C09150=1146.700,365.761,-82.220,-176.299,9.450,148.853
C09151=1146.704,365.478,-82.179,-176.301,9.445,148.852
C09152=1146.709,365.195,-82.139,-176.305,9.440,148.852
C09153=1146.713,364.911,-82.098,-176.307,9.436,148.851
C09154=1146.718,364.628,-82.057,-176.311,9.431,148.851
C09155=1146.722,364.381,-82.022,-176.313,9.427,148.851
C09156=1146.726,364.133,-81.986,-176.316,9.423,148.850
C09157=1146.730,363.886,-81.950,-176.318,9.419,148.850
C09158=1146.734,363.638,-81.915,-176.321,9.415,148.850
C09159=1146.737,363.391,-81.879,-176.323,9.411,148.849
C09160=1146.741,363.144,-81.844,-176.326,9.406,148.849
C09161=1146.745,362.896,-81.808,-176.329,9.402,148.849
C09162=1146.749,362.648,-81.773,-176.331,9.399,148.848
C09163=1146.753,362.401,-81.738,-176.334,9.394,148.848
C09164=1146.757,362.154,-81.703,-176.336,9.390,148.848
C09165=1146.761,361.906,-81.667,-176.339,9.386,148.847
C09166=1146.764,361.659,-81.632,-176.341,9.383,148.847
C09167=1146.768,361.411,-81.597,-176.344,9.379,148.847
C09168=1146.773,361.164,-81.562,-176.347,9.374,148.846
C09169=1146.776,360.917,-81.526,-176.350,9.370,148.846
C09170=1146.780,360.669,-81.490,-176.352,9.367,148.846
C09171=1146.784,360.421,-81.456,-176.354,9.362,148.845
C09172=1146.788,360.174,-81.420,-176.357,9.358,148.845
C09173=1146.792,359.927,-81.385,-176.359,9.355,148.845
C09174=1146.796,359.678,-81.350,-176.362,9.350,148.844
C09175=1146.800,359.432,-81.315,-176.365,9.346,148.844
C09176=1146.804,359.184,-81.280,-176.368,9.342,148.844
C09177=1146.808,358.936,-81.245,-176.369,9.339,148.843
C09178=1146.812,358.689,-81.209,-176.372,9.335,148.843
C09179=1146.816,358.441,-81.175,-176.375,9.330,148.842
C09180=1146.820,358.194,-81.139,-176.377,9.327,148.842
C09181=1146.823,357.947,-81.105,-176.380,9.323,148.842
C09182=1146.827,357.699,-81.070,-176.383,9.318,148.842
C09183=1146.831,357.451,-81.035,-176.385,9.315,148.841
C09184=1146.835,357.204,-81.000,-176.387,9.311,148.841
C09185=1146.839,356.956,-80.965,-176.390,9.306,148.840
C09186=1146.843,356.708,-80.929,-176.392,9.303,148.840
C09187=1146.847,356.461,-80.895,-176.395,9.299,148.840
C09188=1146.850,356.214,-80.860,-176.397,9.295,148.840
C09189=1146.855,355.966,-80.825,-176.400,9.291,148.839
C09190=1146.859,355.719,-80.790,-176.402,9.287,148.839
C09191=1146.863,355.471,-80.755,-176.405,9.284,148.839
C09192=1146.867,355.223,-80.720,-176.407,9.279,148.838
C09193=1146.870,354.976,-80.685,-176.410,9.275,148.838
C09194=1146.875,354.729,-80.651,-176.413,9.272,148.838
C09195=1146.879,354.481,-80.616,-176.415,9.268,148.837
C09196=1146.882,354.233,-80.581,-176.417,9.264,148.837
C09197=1146.886,353.986,-80.547,-176.420,9.260,148.837
C09198=1146.890,353.738,-80.512,-176.423,9.256,148.836
C09199=1146.894,353.491,-80.477,-176.425,9.252,148.836
C09200=1146.898,353.243,-80.442,-176.428,9.248,148.836
C09201=1146.902,352.996,-80.408,-176.431,9.244,148.835
C09202=1146.906,352.748,-80.373,-176.432,9.240,148.835
C09203=1146.910,352.501,-80.338,-176.435,9.236,148.835
C09204=1146.914,352.253,-80.304,-176.437,9.233,148.834
C09205=1146.918,352.006,-80.269,-176.440,9.229,148.834
C09206=1146.922,351.758,-80.234,-176.443,9.225,148.834
C09207=1146.926,351.511,-80.201,-176.445,9.221,148.833
C09208=1146.930,351.263,-80.165,-176.448,9.217,148.833
C09209=1146.934,351.016,-80.131,-176.450,9.213,148.833
C09210=1146.937,350.768,-80.096,-176.453,9.209,148.832
C09211=1146.942,350.520,-80.062,-176.456,9.205,148.832
C09212=1146.946,350.272,-80.027,-176.458,9.202,148.832
C09213=1146.950,350.025,-79.993,-176.460,9.198,148.832
C09214=1146.954,349.777,-79.958,-176.463,9.194,148.831
C09215=1146.958,349.530,-79.924,-176.465,9.190,148.831
C09216=1146.962,349.282,-79.890,-176.468,9.186,148.831
C09217=1146.966,349.034,-79.855,-176.470,9.183,148.830
C09218=1146.969,348.787,-79.821,-176.473,9.178,148.830
C09219=1146.974,348.539,-79.786,-176.475,9.175,148.830
C09220=1146.978,348.292,-79.753,-176.478,9.171,148.830
C09221=1146.982,348.044,-79.718,-176.480,9.167,148.829
C09222=1146.986,347.797,-79.684,-176.483,9.163,148.829
C09223=1146.990,347.549,-79.649,-176.486,9.159,148.829
C09224=1146.993,347.302,-79.615,-176.488,9.155,148.828
C09225=1146.997,347.053,-79.580,-176.491,9.151,148.828
C09226=1147.001,346.806,-79.546,-176.493,9.148,148.828
C09227=1147.006,346.558,-79.513,-176.496,9.144,148.827
C09228=1147.009,346.311,-79.479,-176.498,9.140,148.827
C09229=1147.014,346.063,-79.444,-176.501,9.136,148.827
C09230=1147.018,345.816,-79.410,-176.503,9.132,148.826
C09231=1147.022,345.568,-79.375,-176.506,9.129,148.826
C09232=1147.026,345.321,-79.341,-176.509,9.125,148.826
C09233=1147.030,345.072,-79.307,-176.510,9.121,148.826
C09234=1147.034,344.825,-79.273,-176.513,9.117,148.825
C09235=1147.037,344.578,-79.240,-176.516,9.114,148.825
C09236=1147.042,344.329,-79.205,-176.519,9.110,148.825
C09237=1147.046,344.082,-79.172,-176.520,9.106,148.824
C09238=1147.050,343.835,-79.137,-176.523,9.102,148.824
C09239=1147.053,343.587,-79.103,-176.526,9.098,148.824
C09240=1147.058,343.339,-79.070,-176.528,9.094,148.824
C09241=1147.062,343.092,-79.035,-176.531,9.090,148.823
C09242=1147.066,342.844,-79.001,-176.533,9.087,148.823
C09243=1147.069,342.596,-78.968,-176.536,9.083,148.823
C09244=1147.074,342.349,-78.933,-176.538,9.079,148.822
C09245=1147.078,342.101,-78.900,-176.541,9.075,148.822
C09246=1147.081,341.853,-78.866,-176.544,9.072,148.822
C09247=1147.086,341.606,-78.832,-176.546,9.068,148.822
C09248=1147.090,341.358,-78.798,-176.548,9.064,148.821
C09249=1147.094,341.111,-78.765,-176.551,9.060,148.821
C09250=1147.098,340.862,-78.730,-176.554,9.057,148.821
C09251=1147.102,340.615,-78.697,-176.556,9.053,148.821
C09252=1147.106,340.367,-78.663,-176.558,9.049,148.820
C09253=1147.110,340.120,-78.630,-176.561,9.045,148.820
C09254=1147.114,339.871,-78.595,-176.564,9.041,148.820
C09255=1147.119,339.592,-78.558,-176.567,9.037,148.819
C09256=1147.124,339.311,-78.519,-176.570,9.033,148.819
C09257=1147.128,339.031,-78.481,-176.573,9.028,148.819
C09258=1147.132,338.750,-78.443,-176.575,9.024,148.819
C09259=1147.136,338.503,-78.410,-176.578,9.021,148.818
C09260=1147.140,338.255,-78.376,-176.581,9.017,148.818
C09261=1147.144,338.008,-78.343,-176.583,9.013,148.818
C09262=1147.149,337.760,-78.309,-176.585,9.009,148.817
C09263=1147.153,337.512,-78.275,-176.588,9.005,148.817
C09264=1147.157,337.264,-78.242,-176.591,9.002,148.817
C09265=1147.161,337.016,-78.209,-176.594,8.998,148.817
C09266=1147.165,336.769,-78.175,-176.596,8.995,148.817
C09267=1147.169,336.522,-78.141,-176.598,8.990,148.816
C09268=1147.172,336.273,-78.108,-176.601,8.987,148.816
C09269=1147.176,336.025,-78.075,-176.604,8.983,148.816
C09270=1147.181,335.778,-78.040,-176.606,8.980,148.815
C09271=1147.185,335.530,-78.007,-176.608,8.976,148.815
C09272=1147.189,335.283,-77.974,-176.611,8.972,148.815
C09273=1147.193,335.035,-77.941,-176.613,8.969,148.815
C09274=1147.198,334.787,-77.908,-176.616,8.965,148.814
C09275=1147.201,334.539,-77.874,-176.618,8.961,148.814
C09276=1147.205,334.292,-77.840,-176.621,8.957,148.814
C09277=1147.209,334.044,-77.807,-176.624,8.954,148.814
C09278=1147.213,333.796,-77.774,-176.627,8.950,148.813
C09279=1147.217,333.548,-77.741,-176.629,8.947,148.813
C09280=1147.222,333.301,-77.708,-176.631,8.942,148.813
C09281=1147.226,333.053,-77.675,-176.634,8.939,148.813
C09282=1147.230,332.805,-77.641,-176.637,8.935,148.812
C09283=1147.234,332.557,-77.608,-176.639,8.932,148.812
C09284=1147.237,332.309,-77.575,-176.642,8.928,148.812
C09285=1147.242,332.061,-77.542,-176.644,8.924,148.812
C09286=1147.246,331.814,-77.508,-176.647,8.920,148.812
C09287=1147.250,331.566,-77.475,-176.649,8.917,148.811
C09288=1147.253,331.318,-77.443,-176.652,8.913,148.811
C09289=1147.257,331.071,-77.410,-176.655,8.910,148.811
C09290=1147.262,330.823,-77.376,-176.657,8.906,148.811
C09291=1147.266,330.575,-77.343,-176.659,8.902,148.810
C09292=1147.270,330.327,-77.310,-176.662,8.899,148.810
C09293=1147.274,330.080,-77.277,-176.665,8.895,148.810
C09294=1147.278,329.832,-77.244,-176.667,8.891,148.810
C09295=1147.283,329.584,-77.211,-176.670,8.887,148.809
C09296=1147.287,329.336,-77.178,-176.672,8.884,148.809
C09297=1147.290,329.089,-77.146,-176.675,8.880,148.809
C09298=1147.294,328.841,-77.112,-176.677,8.877,148.809
C09299=1147.298,328.593,-77.079,-176.680,8.872,148.809
C09300=1147.303,328.345,-77.046,-176.683,8.869,148.808
C09301=1147.307,328.097,-77.014,-176.685,8.866,148.808
C09302=1147.310,327.850,-76.981,-176.688,8.862,148.808
C09303=1147.315,327.602,-76.948,-176.690,8.859,148.808
C09304=1147.319,327.354,-76.915,-176.693,8.855,148.807
C09305=1147.323,327.106,-76.882,-176.696,8.851,148.807
C09306=1147.327,326.858,-76.849,-176.698,8.847,148.807
C09307=1147.331,326.611,-76.817,-176.701,8.844,148.807
C09308=1147.335,326.362,-76.784,-176.703,8.841,148.807
C09309=1147.339,326.115,-76.751,-176.706,8.837,148.806
C09310=1147.343,325.867,-76.719,-176.708,8.833,148.806
C09311=1147.347,325.619,-76.686,-176.711,8.829,148.806
C09312=1147.352,325.372,-76.653,-176.714,8.826,148.806
C09313=1147.356,325.123,-76.621,-176.716,8.822,148.806
C09314=1147.360,324.876,-76.588,-176.719,8.819,148.805
C09315=1147.364,324.628,-76.555,-176.721,8.815,148.805
C09316=1147.368,324.380,-76.523,-176.724,8.811,148.805
C09317=1147.372,324.132,-76.490,-176.726,8.808,148.805
C09318=1147.376,323.884,-76.458,-176.729,8.804,148.805
C09319=1147.380,323.636,-76.425,-176.732,8.801,148.804
C09320=1147.384,323.388,-76.393,-176.734,8.797,148.804
C09321=1147.388,323.141,-76.360,-176.737,8.793,148.804
C09322=1147.392,322.893,-76.328,-176.739,8.790,148.804
C09323=1147.396,322.646,-76.295,-176.742,8.786,148.803
C09324=1147.401,322.397,-76.262,-176.744,8.783,148.803
C09325=1147.404,322.150,-76.230,-176.747,8.779,148.803
C09326=1147.409,321.901,-76.197,-176.750,8.775,148.803
C09327=1147.412,321.653,-76.166,-176.752,8.772,148.803
C09328=1147.417,321.406,-76.132,-176.755,8.768,148.802
C09329=1147.421,321.158,-76.101,-176.757,8.765,148.802
C09330=1147.425,320.911,-76.068,-176.760,8.761,148.802
C09331=1147.429,320.663,-76.036,-176.762,8.757,148.802
C09332=1147.433,320.414,-76.004,-176.765,8.754,148.802
C09333=1147.437,320.167,-75.971,-176.768,8.750,148.801
C09334=1147.441,319.918,-75.939,-176.770,8.747,148.801
C09335=1147.445,319.671,-75.907,-176.773,8.744,148.801
C09336=1147.450,319.423,-75.875,-176.776,8.740,148.801
C09337=1147.453,319.175,-75.842,-176.778,8.736,148.801
C09338=1147.458,318.927,-75.810,-176.781,8.732,148.801
C09339=1147.461,318.679,-75.778,-176.783,8.729,148.800
C09340=1147.466,318.431,-75.746,-176.786,8.726,148.800
C09341=1147.470,318.184,-75.713,-176.788,8.722,148.800
C09342=1147.474,317.936,-75.681,-176.791,8.718,148.800
C09343=1147.478,317.687,-75.649,-176.793,8.715,148.800
C09344=1147.482,317.440,-75.617,-176.796,8.711,148.799
C09345=1147.487,317.192,-75.585,-176.799,8.708,148.799
C09346=1147.490,316.944,-75.553,-176.802,8.704,148.799
C09347=1147.495,316.695,-75.521,-176.804,8.701,148.799
C09348=1147.499,316.449,-75.488,-176.806,8.697,148.799
C09349=1147.503,316.201,-75.457,-176.809,8.693,148.799
C09350=1147.507,315.952,-75.424,-176.812,8.690,148.798
C09351=1147.511,315.704,-75.392,-176.814,8.687,148.798
C09352=1147.515,315.457,-75.361,-176.817,8.683,148.798
C09353=1147.519,315.209,-75.328,-176.820,8.680,148.798
C09354=1147.523,314.961,-75.297,-176.822,8.677,148.798
C09355=1147.527,314.713,-75.265,-176.825,8.672,148.798
C09356=1147.532,314.465,-75.233,-176.827,8.669,148.797
C09357=1147.536,314.217,-75.201,-176.830,8.666,148.797
C09358=1147.540,313.969,-75.169,-176.833,8.662,148.797
C09359=1147.545,313.692,-75.133,-176.836,8.658,148.797
C09360=1147.550,313.413,-75.098,-176.838,8.655,148.797
C09361=1147.554,313.136,-75.063,-176.841,8.651,148.797
C09362=1147.558,312.858,-75.027,-176.844,8.647,148.796
C09363=1147.563,312.610,-74.995,-176.847,8.643,148.796
C09364=1147.567,312.363,-74.963,-176.850,8.640,148.796
C09365=1147.571,312.115,-74.931,-176.852,8.636,148.796
C09366=1147.574,311.867,-74.899,-176.855,8.632,148.796
C09367=1147.579,311.619,-74.869,-176.857,8.629,148.796
C09368=1147.583,311.370,-74.836,-176.860,8.626,148.796
C09369=1147.588,311.123,-74.805,-176.863,8.622,148.795
C09370=1147.591,310.875,-74.773,-176.865,8.619,148.795
C09371=1147.596,310.626,-74.742,-176.867,8.615,148.795
C09372=1147.600,310.379,-74.710,-176.870,8.611,148.795
C09373=1147.604,310.131,-74.678,-176.873,8.608,148.795
C09374=1147.609,309.883,-74.646,-176.875,8.605,148.795
C09375=1147.613,309.635,-74.615,-176.878,8.602,148.794
C09376=1147.617,309.387,-74.584,-176.881,8.598,148.794
C09377=1147.621,309.139,-74.552,-176.883,8.595,148.794
C09378=1147.625,308.891,-74.521,-176.886,8.592,148.794
C09379=1147.629,308.643,-74.489,-176.889,8.587,148.794
C09380=1147.633,308.395,-74.457,-176.891,8.584,148.794
C09381=1147.637,308.147,-74.427,-176.894,8.581,148.794
C09382=1147.642,307.899,-74.394,-176.897,8.577,148.793
C09383=1147.646,307.651,-74.363,-176.899,8.574,148.793
C09384=1147.650,307.403,-74.332,-176.901,8.571,148.793
C09385=1147.654,307.156,-74.300,-176.905,8.567,148.793
C09386=1147.658,306.907,-74.269,-176.907,8.564,148.793
C09387=1147.663,306.660,-74.238,-176.909,8.560,148.793
C09388=1147.667,306.411,-74.206,-176.912,8.557,148.793
C09389=1147.671,306.164,-74.175,-176.915,8.553,148.793
C09390=1147.675,305.915,-74.144,-176.917,8.550,148.792
C09391=1147.679,305.668,-74.112,-176.920,8.547,148.792
C09392=1147.683,305.419,-74.081,-176.923,8.543,148.792
C09393=1147.688,305.172,-74.050,-176.925,8.540,148.792
C09394=1147.692,304.923,-74.019,-176.928,8.536,148.792
C09395=1147.696,304.675,-73.988,-176.930,8.534,148.792
C09396=1147.700,304.427,-73.956,-176.933,8.529,148.792
C09397=1147.705,304.179,-73.925,-176.936,8.526,148.791
C09398=1147.708,303.931,-73.893,-176.938,8.523,148.791
C09399=1147.713,303.683,-73.863,-176.941,8.519,148.791
C09400=1147.717,303.435,-73.832,-176.944,8.516,148.791
C09401=1147.720,303.187,-73.801,-176.946,8.513,148.791
C09402=1147.725,302.939,-73.770,-176.949,8.510,148.791
C09403=1147.729,302.691,-73.739,-176.952,8.506,148.791
C09404=1147.733,302.443,-73.707,-176.954,8.503,148.791
C09405=1147.738,302.195,-73.676,-176.957,8.499,148.791
C09406=1147.742,301.947,-73.645,-176.960,8.495,148.790
C09407=1147.747,301.699,-73.615,-176.963,8.492,148.790
C09408=1147.750,301.451,-73.583,-176.965,8.489,148.790
C09409=1147.754,301.203,-73.553,-176.967,8.486,148.790
C09410=1147.759,300.955,-73.522,-176.971,8.482,148.790
C09411=1147.763,300.706,-73.491,-176.973,8.479,148.790
C09412=1147.767,300.459,-73.460,-176.976,8.476,148.790
C09413=1147.771,300.210,-73.428,-176.978,8.473,148.790
C09414=1147.775,299.963,-73.398,-176.981,8.468,148.789
C09415=1147.780,299.715,-73.367,-176.984,8.466,148.789
C09416=1147.784,299.466,-73.336,-176.986,8.462,148.789
C09417=1147.788,299.218,-73.305,-176.988,8.459,148.789
C09418=1147.792,298.971,-73.275,-176.992,8.455,148.789
C09419=1147.796,298.722,-73.244,-176.994,8.452,148.789
C09420=1147.801,298.474,-73.213,-176.997,8.449,148.789
C09421=1147.805,298.226,-73.182,-176.999,8.446,148.789
C09422=1147.809,297.978,-73.152,-177.002,8.442,148.789
C09423=1147.813,297.730,-73.121,-177.005,8.439,148.789
C09424=1147.818,297.482,-73.090,-177.007,8.435,148.788
C09425=1147.822,297.233,-73.059,-177.010,8.433,148.788
C09426=1147.826,296.985,-73.029,-177.013,8.428,148.788
C09427=1147.830,296.737,-72.998,-177.015,8.425,148.788
C09428=1147.835,296.490,-72.967,-177.018,8.422,148.788
C09429=1147.838,296.241,-72.937,-177.020,8.419,148.788
C09430=1147.843,295.993,-72.906,-177.023,8.416,148.788
C09431=1147.847,295.746,-72.876,-177.026,8.412,148.788
C09432=1147.851,295.497,-72.845,-177.029,8.409,148.788
C09433=1147.855,295.249,-72.814,-177.031,8.406,148.788
C09434=1147.859,295.001,-72.784,-177.034,8.403,148.788
C09435=1147.864,294.753,-72.753,-177.037,8.399,148.787
C09436=1147.867,294.505,-72.723,-177.039,8.396,148.788
C09437=1147.872,294.256,-72.693,-177.042,8.392,148.787
C09438=1147.877,294.008,-72.662,-177.044,8.390,148.787
C09439=1147.881,293.761,-72.632,-177.047,8.386,148.787
C09440=1147.885,293.512,-72.601,-177.050,8.382,148.787
C09441=1147.888,293.265,-72.570,-177.052,8.379,148.787
C09442=1147.893,293.016,-72.540,-177.055,8.376,148.787
C09443=1147.897,292.768,-72.510,-177.058,8.373,148.787
C09444=1147.902,292.520,-72.479,-177.060,8.369,148.787
C09445=1147.905,292.271,-72.450,-177.063,8.366,148.787
C09446=1147.910,292.023,-72.419,-177.066,8.363,148.787
C09447=1147.914,291.776,-72.389,-177.068,8.360,148.787
C09448=1147.919,291.528,-72.358,-177.071,8.357,148.786
C09449=1147.923,291.280,-72.328,-177.074,8.353,148.786
C09450=1147.927,291.031,-72.297,-177.076,8.350,148.786
C09451=1147.931,290.783,-72.268,-177.079,8.347,148.786
C09452=1147.935,290.535,-72.238,-177.081,8.343,148.786
C09453=1147.939,290.287,-72.207,-177.084,8.340,148.786
C09454=1147.944,290.039,-72.177,-177.087,8.336,148.786
C09455=1147.948,289.791,-72.147,-177.090,8.333,148.786
C09456=1147.952,289.543,-72.117,-177.093,8.330,148.786
C09457=1147.956,289.294,-72.086,-177.095,8.327,148.786
C09458=1147.960,289.046,-72.056,-177.098,8.324,148.786
C09459=1147.964,288.798,-72.026,-177.100,8.321,148.786
C09460=1147.969,288.550,-71.996,-177.103,8.317,148.786
C09461=1147.973,288.302,-71.966,-177.106,8.314,148.786
C09462=1147.977,288.054,-71.936,-177.109,8.311,148.786
C09463=1147.982,287.778,-71.903,-177.111,8.307,148.785
C09464=1147.987,287.503,-71.869,-177.114,8.304,148.785
C09465=1147.992,287.228,-71.837,-177.118,8.300,148.785
C09466=1147.996,286.952,-71.803,-177.121,8.296,148.785
C09467=1148.001,286.703,-71.773,-177.123,8.293,148.785
C09468=1148.005,286.456,-71.743,-177.126,8.290,148.785
C09469=1148.009,286.208,-71.713,-177.128,8.287,148.785
C09470=1148.013,285.959,-71.684,-177.131,8.284,148.785
C09471=1148.018,285.711,-71.653,-177.133,8.281,148.785
C09472=1148.022,285.463,-71.624,-177.137,8.277,148.785
C09473=1148.026,285.215,-71.594,-177.139,8.274,148.785
C09474=1148.031,284.967,-71.563,-177.142,8.271,148.785
C09475=1148.035,284.719,-71.534,-177.144,8.267,148.785
C09476=1148.039,284.470,-71.504,-177.147,8.265,148.785
C09477=1148.043,284.223,-71.474,-177.150,8.262,148.785
C09478=1148.047,283.974,-71.445,-177.153,8.258,148.785
C09479=1148.052,283.726,-71.415,-177.155,8.255,148.785
C09480=1148.056,283.478,-71.385,-177.158,8.251,148.785
C09481=1148.060,283.229,-71.356,-177.161,8.248,148.785
C09482=1148.064,282.982,-71.326,-177.163,8.245,148.785
C09483=1148.068,282.733,-71.296,-177.166,8.242,148.784
C09484=1148.073,282.485,-71.266,-177.168,8.239,148.784
C09485=1148.077,282.237,-71.237,-177.172,8.235,148.784
C09486=1148.082,281.988,-71.207,-177.174,8.232,148.784
C09487=1148.086,281.740,-71.178,-177.177,8.229,148.784
C09488=1148.090,281.492,-71.148,-177.179,8.226,148.784
C09489=1148.094,281.244,-71.118,-177.182,8.223,148.784
C09490=1148.098,280.996,-71.089,-177.185,8.220,148.784
C09491=1148.102,280.748,-71.059,-177.187,8.217,148.784
C09492=1148.107,280.499,-71.029,-177.190,8.213,148.784
C09493=1148.111,280.251,-71.000,-177.193,8.210,148.784
C09494=1148.116,280.003,-70.971,-177.196,8.207,148.784
C09495=1148.120,279.755,-70.941,-177.198,8.204,148.784
C09496=1148.124,279.507,-70.912,-177.201,8.201,148.784
C09497=1148.129,279.258,-70.882,-177.203,8.198,148.784
C09498=1148.133,279.010,-70.853,-177.206,8.195,148.784
C09499=1148.137,278.762,-70.823,-177.209,8.192,148.784
C09500=1148.141,278.514,-70.794,-177.212,8.188,148.784
C09501=1148.145,278.265,-70.765,-177.215,8.185,148.784
C09502=1148.150,278.017,-70.735,-177.217,8.182,148.784
C09503=1148.154,277.768,-70.706,-177.220,8.179,148.784
C09504=1148.159,277.521,-70.677,-177.223,8.176,148.784
C09505=1148.163,277.272,-70.648,-177.225,8.173,148.784
C09506=1148.167,277.024,-70.618,-177.228,8.170,148.784
C09507=1148.171,276.776,-70.589,-177.230,8.167,148.784
C09508=1148.176,276.527,-70.559,-177.233,8.164,148.784
C09509=1148.180,276.279,-70.530,-177.237,8.160,148.784
C09510=1148.183,276.031,-70.502,-177.239,8.157,148.784
C09511=1148.188,275.783,-70.473,-177.242,8.154,148.784
C09512=1148.192,275.535,-70.443,-177.244,8.151,148.784
C09513=1148.197,275.287,-70.414,-177.247,8.147,148.784
C09514=1148.201,275.038,-70.384,-177.250,8.145,148.784
C09515=1148.205,274.789,-70.356,-177.252,8.142,148.784
C09516=1148.209,274.541,-70.326,-177.255,8.139,148.784
C09517=1148.214,274.294,-70.297,-177.257,8.135,148.784
C09518=1148.219,274.045,-70.268,-177.260,8.132,148.784
C09519=1148.222,273.797,-70.240,-177.264,8.129,148.784
C09520=1148.226,273.548,-70.210,-177.266,8.125,148.784
C09521=1148.231,273.300,-70.181,-177.269,8.122,148.784
C09522=1148.236,273.052,-70.152,-177.271,8.120,148.784
C09523=1148.240,272.804,-70.123,-177.274,8.117,148.784
C09524=1148.244,272.555,-70.095,-177.277,8.113,148.784
C09525=1148.248,272.307,-70.065,-177.279,8.110,148.784
C09526=1148.253,272.059,-70.037,-177.282,8.107,148.784
C09527=1148.257,271.810,-70.007,-177.285,8.105,148.784
C09528=1148.261,271.562,-69.978,-177.287,8.101,148.784
C09529=1148.265,271.314,-69.950,-177.290,8.098,148.784
C09530=1148.270,271.066,-69.921,-177.293,8.095,148.784
C09531=1148.274,270.817,-69.892,-177.296,8.092,148.784
C09532=1148.278,270.569,-69.863,-177.298,8.088,148.784
C09533=1148.282,270.320,-69.834,-177.301,8.085,148.784
C09534=1148.287,270.073,-69.805,-177.304,8.083,148.784
C09535=1148.291,269.824,-69.777,-177.307,8.080,148.784
C09536=1148.295,269.576,-69.748,-177.310,8.077,148.784
C09537=1148.300,269.328,-69.719,-177.312,8.073,148.784
C09538=1148.304,269.079,-69.691,-177.315,8.070,148.784
C09539=1148.308,268.831,-69.662,-177.317,8.068,148.784
C09540=1148.313,268.583,-69.633,-177.320,8.065,148.784
C09541=1148.317,268.334,-69.604,-177.323,8.062,148.784
C09542=1148.321,268.086,-69.576,-177.325,8.058,148.784
C09543=1148.326,267.838,-69.547,-177.328,8.055,148.784
C09544=1148.330,267.589,-69.518,-177.331,8.052,148.784
C09545=1148.334,267.341,-69.490,-177.334,8.050,148.784
C09546=1148.339,267.093,-69.461,-177.336,8.047,148.784
C09547=1148.342,266.845,-69.433,-177.339,8.043,148.784
C09548=1148.347,266.596,-69.404,-177.342,8.040,148.784
C09549=1148.352,266.348,-69.375,-177.345,8.037,148.784
C09550=1148.356,266.099,-69.347,-177.348,8.034,148.784
C09551=1148.361,265.851,-69.318,-177.350,8.031,148.784
C09552=1148.364,265.603,-69.290,-177.353,8.028,148.784
C09553=1148.369,265.354,-69.261,-177.356,8.025,148.784
C09554=1148.373,265.106,-69.234,-177.358,8.022,148.784
C09555=1148.378,264.857,-69.205,-177.361,8.019,148.784
C09556=1148.382,264.610,-69.176,-177.364,8.016,148.784
C09557=1148.386,264.361,-69.148,-177.367,8.013,148.784
C09558=1148.391,264.113,-69.119,-177.370,8.010,148.784
C09559=1148.395,263.864,-69.091,-177.372,8.007,148.784
C09560=1148.399,263.615,-69.062,-177.375,8.004,148.784
C09561=1148.404,263.367,-69.035,-177.377,8.001,148.784
C09562=1148.408,263.119,-69.006,-177.380,7.998,148.784
C09563=1148.413,262.871,-68.978,-177.383,7.995,148.784
C09564=1148.416,262.622,-68.950,-177.386,7.992,148.784
C09565=1148.421,262.375,-68.921,-177.389,7.989,148.784
C09566=1148.425,262.126,-68.893,-177.391,7.986,148.784
C09567=1148.430,261.852,-68.861,-177.394,7.983,148.784
C09568=1148.435,261.579,-68.831,-177.397,7.979,148.784
C09569=1148.440,261.306,-68.800,-177.400,7.976,148.784
C09570=1148.445,261.032,-68.769,-177.403,7.972,148.784
C09571=1148.449,260.783,-68.741,-177.406,7.970,148.784
C09572=1148.453,260.536,-68.713,-177.409,7.967,148.784
C09573=1148.458,260.287,-68.684,-177.411,7.964,148.785
C09574=1148.462,260.039,-68.656,-177.414,7.961,148.785
C09575=1148.466,259.790,-68.628,-177.417,7.958,148.785
C09576=1148.471,259.542,-68.600,-177.420,7.955,148.785
C09577=1148.475,259.293,-68.572,-177.423,7.952,148.785
C09578=1148.479,259.046,-68.544,-177.425,7.949,148.785
C09579=1148.483,258.797,-68.515,-177.428,7.946,148.785
C09580=1148.488,258.548,-68.488,-177.430,7.943,148.785
C09581=1148.492,258.300,-68.460,-177.433,7.940,148.785
C09582=1148.497,258.051,-68.432,-177.436,7.937,148.785
C09583=1148.501,257.803,-68.403,-177.439,7.934,148.785
C09584=1148.505,257.555,-68.376,-177.442,7.931,148.785
C09585=1148.510,257.307,-68.349,-177.444,7.928,148.785
C09586=1148.514,257.058,-68.320,-177.447,7.925,148.785
C09587=1148.519,256.810,-68.292,-177.450,7.922,148.785
C09588=1148.522,256.561,-68.264,-177.453,7.919,148.785
C09589=1148.527,256.313,-68.237,-177.456,7.916,148.785
C09590=1148.531,256.064,-68.208,-177.458,7.913,148.785
C09591=1148.536,255.816,-68.180,-177.461,7.910,148.785
C09592=1148.540,255.567,-68.153,-177.463,7.907,148.785
C09593=1148.544,255.319,-68.125,-177.466,7.904,148.785
C09594=1148.549,255.071,-68.097,-177.468,7.902,148.785
C09595=1148.554,254.822,-68.070,-177.471,7.899,148.786
C09596=1148.558,254.574,-68.042,-177.474,7.896,148.786
C09597=1148.562,254.326,-68.014,-177.477,7.893,148.786
C09598=1148.566,254.077,-67.986,-177.480,7.890,148.786
C09599=1148.570,253.829,-67.959,-177.482,7.888,148.786
C09600=1148.575,253.580,-67.932,-177.485,7.885,148.786
C09601=1148.579,253.332,-67.903,-177.488,7.882,148.786
C09602=1148.584,253.083,-67.876,-177.491,7.879,148.786
C09603=1148.589,252.835,-67.848,-177.493,7.876,148.786
C09604=1148.592,252.586,-67.820,-177.496,7.873,148.786
C09605=1148.597,252.338,-67.793,-177.499,7.870,148.786
C09606=1148.601,252.090,-67.765,-177.502,7.867,148.786
C09607=1148.605,251.841,-67.738,-177.505,7.864,148.786
C09608=1148.610,251.592,-67.710,-177.507,7.861,148.786
C09609=1148.614,251.344,-67.683,-177.510,7.858,148.786
C09610=1148.619,251.096,-67.656,-177.513,7.855,148.787
C09611=1148.623,250.847,-67.628,-177.516,7.852,148.787
C09612=1148.627,250.599,-67.600,-177.518,7.849,148.787
C09613=1148.632,250.351,-67.573,-177.521,7.847,148.787
C09614=1148.636,250.102,-67.545,-177.524,7.844,148.787
C09615=1148.641,249.853,-67.518,-177.527,7.841,148.787
C09616=1148.645,249.605,-67.490,-177.529,7.839,148.787
C09617=1148.650,249.357,-67.463,-177.532,7.836,148.787
C09618=1148.654,249.108,-67.436,-177.535,7.833,148.787
C09619=1148.658,248.860,-67.408,-177.537,7.830,148.787
C09620=1148.663,248.611,-67.381,-177.540,7.827,148.787
C09621=1148.667,248.363,-67.354,-177.543,7.824,148.787
C09622=1148.671,248.114,-67.326,-177.546,7.821,148.787
C09623=1148.676,247.866,-67.299,-177.549,7.818,148.787
C09624=1148.680,247.617,-67.272,-177.551,7.815,148.788
C09625=1148.685,247.369,-67.245,-177.554,7.812,148.788
C09626=1148.690,247.120,-67.218,-177.557,7.809,148.788
C09627=1148.693,246.872,-67.190,-177.560,7.806,148.788
C09628=1148.697,246.623,-67.163,-177.562,7.803,148.788
C09629=1148.702,246.375,-67.136,-177.565,7.801,148.788
C09630=1148.707,246.126,-67.109,-177.567,7.798,148.788
C09631=1148.711,245.878,-67.082,-177.570,7.795,148.788
C09632=1148.715,245.629,-67.054,-177.573,7.793,148.788
C09633=1148.720,245.381,-67.027,-177.576,7.790,148.788
C09634=1148.724,245.133,-67.000,-177.579,7.787,148.788
C09635=1148.728,244.884,-66.973,-177.581,7.784,148.788
C09636=1148.733,244.636,-66.946,-177.584,7.781,148.788
C09637=1148.738,244.387,-66.919,-177.587,7.778,148.789
C09638=1148.742,244.138,-66.892,-177.590,7.775,148.789
C09639=1148.746,243.890,-66.865,-177.593,7.772,148.789
C09640=1148.750,243.641,-66.838,-177.595,7.770,148.789
C09641=1148.755,243.393,-66.811,-177.598,7.767,148.789
C09642=1148.760,243.144,-66.784,-177.601,7.764,148.789
C09643=1148.764,242.896,-66.757,-177.604,7.761,148.789
C09644=1148.768,242.648,-66.730,-177.606,7.759,148.789
C09645=1148.773,242.399,-66.703,-177.609,7.756,148.789
C09646=1148.777,242.150,-66.676,-177.612,7.753,148.789
C09647=1148.781,241.902,-66.649,-177.615,7.750,148.790
C09648=1148.785,241.653,-66.622,-177.617,7.747,148.790
C09649=1148.790,241.405,-66.595,-177.620,7.745,148.790
C09650=1148.795,241.156,-66.568,-177.622,7.742,148.790
C09651=1148.799,240.908,-66.542,-177.625,7.739,148.790
C09652=1148.803,240.660,-66.515,-177.628,7.736,148.790
C09653=1148.808,240.411,-66.488,-177.631,7.733,148.790
C09654=1148.812,240.162,-66.462,-177.634,7.730,148.790
C09655=1148.817,239.914,-66.435,-177.637,7.727,148.790
C09656=1148.821,239.665,-66.408,-177.640,7.725,148.790
C09657=1148.825,239.417,-66.381,-177.642,7.722,148.791
C09658=1148.830,239.169,-66.354,-177.645,7.720,148.791
C09659=1148.834,238.920,-66.328,-177.647,7.717,148.791
C09660=1148.839,238.671,-66.301,-177.650,7.714,148.791
C09661=1148.844,238.423,-66.274,-177.653,7.711,148.791
C09662=1148.847,238.175,-66.248,-177.656,7.708,148.791
C09663=1148.852,237.926,-66.222,-177.659,7.705,148.791
C09664=1148.856,237.677,-66.195,-177.661,7.703,148.791
C09665=1148.861,237.429,-66.168,-177.664,7.700,148.791
C09666=1148.866,237.180,-66.142,-177.667,7.697,148.792
C09667=1148.870,236.932,-66.115,-177.670,7.694,148.792
C09668=1148.875,236.683,-66.088,-177.672,7.691,148.792
C09669=1148.879,236.434,-66.062,-177.675,7.688,148.792
C09670=1148.883,236.186,-66.035,-177.678,7.686,148.792
C09671=1148.887,235.914,-66.006,-177.681,7.683,148.792
C09672=1148.893,235.642,-65.978,-177.684,7.680,148.792
C09673=1148.898,235.370,-65.948,-177.687,7.677,148.792
C09674=1148.902,235.099,-65.919,-177.690,7.675,148.793
C09675=1148.907,234.850,-65.893,-177.693,7.672,148.793
C09676=1148.911,234.601,-65.867,-177.696,7.669,148.793
C09677=1148.915,234.353,-65.841,-177.698,7.666,148.793
C09678=1148.920,234.104,-65.814,-177.701,7.663,148.793
C09679=1148.924,233.855,-65.788,-177.704,7.660,148.793
C09680=1148.929,233.607,-65.761,-177.707,7.658,148.793
C09681=1148.933,233.358,-65.735,-177.709,7.655,148.793
C09682=1148.938,233.110,-65.709,-177.712,7.652,148.794
C09683=1148.943,232.861,-65.683,-177.715,7.649,148.794
C09684=1148.946,232.613,-65.656,-177.718,7.646,148.794
C09685=1148.951,232.364,-65.630,-177.720,7.644,148.794
C09686=1148.955,232.116,-65.604,-177.723,7.642,148.794
C09687=1148.960,231.867,-65.577,-177.726,7.639,148.794
C09688=1148.965,231.618,-65.551,-177.729,7.636,148.794
C09689=1148.968,231.370,-65.525,-177.732,7.633,148.794
C09690=1148.973,231.121,-65.499,-177.734,7.631,148.794
C09691=1148.978,230.873,-65.473,-177.737,7.628,148.795
C09692=1148.982,230.624,-65.447,-177.740,7.625,148.795
C09693=1148.987,230.375,-65.420,-177.743,7.622,148.795
C09694=1148.991,230.127,-65.395,-177.745,7.620,148.795
C09695=1148.995,229.878,-65.368,-177.748,7.617,148.795
C09696=1149.000,229.629,-65.342,-177.750,7.614,148.795
C09697=1149.005,229.381,-65.317,-177.754,7.612,148.796
C09698=1149.009,229.133,-65.290,-177.756,7.609,148.796
C09699=1149.013,228.884,-65.264,-177.759,7.606,148.796
C09700=1149.018,228.635,-65.238,-177.761,7.604,148.796
C09701=1149.022,228.386,-65.212,-177.764,7.601,148.796
C09702=1149.027,228.138,-65.187,-177.768,7.598,148.796
C09703=1149.031,227.890,-65.160,-177.770,7.596,148.796
C09704=1149.036,227.641,-65.134,-177.773,7.593,148.796
C09705=1149.040,227.392,-65.108,-177.775,7.590,148.796
C09706=1149.045,227.143,-65.082,-177.779,7.588,148.797
C09707=1149.049,226.895,-65.057,-177.781,7.585,148.797
C09708=1149.054,226.646,-65.031,-177.784,7.582,148.797
C09709=1149.058,226.398,-65.004,-177.787,7.579,148.797
C09710=1149.062,226.149,-64.979,-177.789,7.577,148.797
C09711=1149.067,225.901,-64.953,-177.792,7.574,148.797
C09712=1149.072,225.652,-64.927,-177.795,7.572,148.798
C09713=1149.076,225.403,-64.902,-177.798,7.569,148.798
C09714=1149.080,225.154,-64.876,-177.800,7.567,148.798
C09715=1149.085,224.906,-64.851,-177.803,7.564,148.798
C09716=1149.090,224.657,-64.824,-177.806,7.561,148.798
C09717=1149.094,224.408,-64.798,-177.809,7.558,148.798
C09718=1149.098,224.160,-64.773,-177.811,7.556,148.798
C09719=1149.103,223.912,-64.747,-177.814,7.553,148.799
C09720=1149.107,223.663,-64.722,-177.817,7.550,148.799
C09721=1149.111,223.414,-64.696,-177.820,7.548,148.799
C09722=1149.116,223.166,-64.670,-177.822,7.545,148.799
C09723=1149.121,222.917,-64.645,-177.826,7.543,148.799
C09724=1149.125,222.668,-64.619,-177.828,7.540,148.799
C09725=1149.130,222.420,-64.594,-177.831,7.537,148.799
C09726=1149.134,222.171,-64.568,-177.833,7.535,148.800
C09727=1149.138,221.922,-64.542,-177.837,7.532,148.800
C09728=1149.143,221.674,-64.517,-177.839,7.529,148.800
C09729=1149.147,221.425,-64.492,-177.842,7.527,148.800
C09730=1149.152,221.176,-64.466,-177.845,7.525,148.800
C09731=1149.156,220.928,-64.440,-177.848,7.522,148.800
C09732=1149.161,220.679,-64.415,-177.850,7.519,148.801
C09733=1149.165,220.430,-64.389,-177.853,7.517,148.801
C09734=1149.170,220.182,-64.364,-177.856,7.514,148.801
C09735=1149.174,219.933,-64.339,-177.859,7.511,148.801
C09736=1149.179,219.685,-64.313,-177.861,7.508,148.801
C09737=1149.183,219.436,-64.287,-177.864,7.507,148.802
C09738=1149.188,219.187,-64.262,-177.867,7.504,148.802
C09739=1149.193,218.938,-64.237,-177.870,7.501,148.802
C09740=1149.197,218.690,-64.211,-177.872,7.499,148.802
C09741=1149.201,218.441,-64.185,-177.875,7.496,148.802
C09742=1149.206,218.192,-64.161,-177.878,7.493,148.802
C09743=1149.210,217.943,-64.135,-177.881,7.490,148.802
C09744=1149.215,217.696,-64.110,-177.883,7.489,148.803
C09745=1149.219,217.446,-64.085,-177.886,7.486,148.803
C09746=1149.224,217.198,-64.060,-177.889,7.483,148.803
C09747=1149.228,216.949,-64.034,-177.892,7.481,148.803
C09748=1149.233,216.700,-64.009,-177.895,7.478,148.803
C09749=1149.237,216.452,-63.984,-177.897,7.475,148.803
C09750=1149.242,216.202,-63.959,-177.901,7.472,148.804
C09751=1149.246,215.954,-63.934,-177.903,7.470,148.804
C09752=1149.251,215.705,-63.909,-177.906,7.467,148.804
C09753=1149.255,215.457,-63.883,-177.909,7.465,148.804
C09754=1149.260,215.208,-63.858,-177.911,7.463,148.804
C09755=1149.265,214.959,-63.833,-177.914,7.460,148.804
C09756=1149.268,214.711,-63.808,-177.917,7.457,148.805
C09757=1149.273,214.462,-63.783,-177.919,7.455,148.805
C09758=1149.278,214.213,-63.757,-177.922,7.452,148.805
C09759=1149.283,213.965,-63.733,-177.925,7.450,148.805
C09760=1149.286,213.716,-63.708,-177.928,7.448,148.805
C09761=1149.291,213.467,-63.683,-177.930,7.445,148.806
C09762=1149.296,213.218,-63.658,-177.934,7.442,148.806
C09763=1149.301,212.970,-63.633,-177.936,7.440,148.806
C09764=1149.305,212.721,-63.608,-177.939,7.437,148.806
C09765=1149.309,212.473,-63.583,-177.942,7.435,148.806
C09766=1149.314,212.223,-63.558,-177.944,7.432,148.806
C09767=1149.318,211.975,-63.534,-177.947,7.429,148.807
C09768=1149.323,211.726,-63.508,-177.950,7.427,148.807
C09769=1149.328,211.477,-63.483,-177.952,7.425,148.807
C09770=1149.332,211.229,-63.459,-177.956,7.422,148.807
C09771=1149.336,210.980,-63.433,-177.958,7.419,148.807
C09772=1149.341,210.731,-63.409,-177.961,7.417,148.808
C09773=1149.345,210.482,-63.384,-177.964,7.415,148.808
C09774=1149.350,210.234,-63.359,-177.966,7.413,148.808
C09775=1149.355,209.963,-63.332,-177.969,7.410,148.808
C09776=1149.360,209.693,-63.305,-177.972,7.407,148.808
C09777=1149.364,209.422,-63.278,-177.975,7.404,148.809
C09778=1149.369,209.152,-63.251,-177.978,7.402,148.809
C09779=1149.374,208.903,-63.226,-177.982,7.399,148.809
C09780=1149.379,208.654,-63.202,-177.984,7.396,148.809
C09781=1149.383,208.406,-63.177,-177.987,7.394,148.809
C09782=1149.388,208.156,-63.152,-177.990,7.391,148.810
C09783=1149.392,207.908,-63.128,-177.992,7.389,148.810
C09784=1149.397,207.660,-63.103,-177.995,7.387,148.810
C09785=1149.401,207.410,-63.079,-177.998,7.384,148.810
C09786=1149.406,207.162,-63.054,-178.000,7.382,148.810
C09787=1149.411,206.913,-63.030,-178.004,7.379,148.811
C09788=1149.415,206.664,-63.005,-178.006,7.376,148.811
C09789=1149.419,206.416,-62.981,-178.009,7.374,148.811
C09790=1149.425,206.167,-62.956,-178.012,7.372,148.811
C09791=1149.428,205.918,-62.932,-178.014,7.369,148.811
C09792=1149.434,205.669,-62.907,-178.017,7.367,148.812
C09793=1149.438,205.421,-62.883,-178.020,7.364,148.812
C09794=1149.442,205.171,-62.858,-178.023,7.362,148.812
C09795=1149.447,204.923,-62.834,-178.026,7.359,148.812
C09796=1149.452,204.674,-62.809,-178.028,7.358,148.813
C09797=1149.456,204.425,-62.785,-178.031,7.355,148.813
C09798=1149.461,204.176,-62.760,-178.034,7.352,148.813
C09799=1149.465,203.928,-62.736,-178.037,7.350,148.813
C09800=1149.470,203.679,-62.712,-178.039,7.347,148.813
C09801=1149.474,203.430,-62.687,-178.042,7.345,148.814
C09802=1149.479,203.181,-62.663,-178.045,7.342,148.814
C09803=1149.484,202.933,-62.638,-178.048,7.340,148.814
C09804=1149.488,202.684,-62.614,-178.050,7.338,148.814
C09805=1149.492,202.435,-62.590,-178.054,7.335,148.815
C09806=1149.497,202.187,-62.565,-178.056,7.333,148.815
C09807=1149.501,201.938,-62.541,-178.059,7.331,148.815
C09808=1149.506,201.688,-62.517,-178.062,7.328,148.815
C09809=1149.511,201.440,-62.492,-178.064,7.326,148.815
C09810=1149.515,201.191,-62.468,-178.067,7.323,148.816
C09811=1149.519,200.943,-62.444,-178.070,7.321,148.816
C09812=1149.525,200.694,-62.420,-178.073,7.318,148.816
C09813=1149.528,200.445,-62.395,-178.075,7.316,148.816
C09814=1149.533,200.196,-62.372,-178.078,7.314,148.816
C09815=1149.538,199.948,-62.348,-178.080,7.312,148.817
C09816=1149.543,199.699,-62.323,-178.084,7.309,148.817
C09817=1149.547,199.450,-62.299,-178.087,7.306,148.817
C09818=1149.551,199.201,-62.275,-178.089,7.304,148.817
C09819=1149.556,198.952,-62.251,-178.092,7.301,148.817
C09820=1149.561,198.704,-62.226,-178.095,7.300,148.818
C09821=1149.565,198.454,-62.203,-178.098,7.297,148.818
C09822=1149.570,198.206,-62.179,-178.100,7.295,148.818
C09823=1149.574,197.957,-62.155,-178.103,7.292,148.818
C09824=1149.579,197.708,-62.131,-178.106,7.290,148.819
C09825=1149.583,197.459,-62.107,-178.108,7.287,148.819
C09826=1149.588,197.211,-62.082,-178.112,7.285,148.819
C09827=1149.592,196.962,-62.059,-178.114,7.283,148.819
C09828=1149.597,196.713,-62.035,-178.117,7.280,148.820
C09829=1149.602,196.464,-62.011,-178.119,7.278,148.820
C09830=1149.606,196.215,-61.987,-178.123,7.275,148.820
C09831=1149.610,195.966,-61.963,-178.125,7.273,148.820
C09832=1149.615,195.717,-61.939,-178.128,7.271,148.821
C09833=1149.620,195.469,-61.915,-178.131,7.269,148.821
C09834=1149.624,195.220,-61.892,-178.134,7.266,148.821
C09835=1149.629,194.972,-61.868,-178.136,7.264,148.821
C09836=1149.633,194.723,-61.844,-178.139,7.262,148.821
C09837=1149.639,194.474,-61.820,-178.142,7.260,148.822
C09838=1149.643,194.225,-61.796,-178.145,7.257,148.822
C09839=1149.648,193.976,-61.772,-178.147,7.255,148.822
C09840=1149.652,193.727,-61.749,-178.150,7.252,148.822
C09841=1149.656,193.478,-61.725,-178.153,7.250,148.823
C09842=1149.661,193.229,-61.701,-178.156,7.248,148.823
C09843=1149.665,192.980,-61.678,-178.159,7.245,148.823
C09844=1149.670,192.732,-61.654,-178.161,7.243,148.823
C09845=1149.675,192.483,-61.630,-178.164,7.240,148.824
C09846=1149.679,192.234,-61.607,-178.167,7.239,148.824
C09847=1149.684,191.985,-61.583,-178.170,7.236,148.824
C09848=1149.688,191.736,-61.560,-178.173,7.234,148.825
C09849=1149.693,191.488,-61.535,-178.175,7.231,148.825
C09850=1149.697,191.239,-61.512,-178.178,7.229,148.825
C09851=1149.702,190.990,-61.489,-178.181,7.226,148.825
C09852=1149.707,190.741,-61.465,-178.184,7.225,148.825
C09853=1149.711,190.492,-61.441,-178.187,7.222,148.826
C09854=1149.716,190.243,-61.418,-178.189,7.220,148.826
C09855=1149.721,189.994,-61.395,-178.192,7.217,148.826
C09856=1149.725,189.746,-61.371,-178.195,7.215,148.826
C09857=1149.730,189.497,-61.347,-178.197,7.214,148.827
C09858=1149.734,189.248,-61.324,-178.200,7.211,148.827
C09859=1149.739,188.999,-61.300,-178.203,7.209,148.827
C09860=1149.744,188.750,-61.277,-178.206,7.206,148.828
C09861=1149.748,188.501,-61.253,-178.208,7.204,148.828
C09862=1149.753,188.252,-61.230,-178.211,7.202,148.828
C09863=1149.757,188.004,-61.207,-178.214,7.200,148.828
C09864=1149.762,187.755,-61.184,-178.217,7.197,148.829
C09865=1149.767,187.506,-61.161,-178.220,7.195,148.829
C09866=1149.772,187.257,-61.137,-178.222,7.192,148.829
C09867=1149.776,187.008,-61.114,-178.225,7.191,148.829
C09868=1149.781,186.760,-61.090,-178.228,7.188,148.829
C09869=1149.785,186.511,-61.066,-178.231,7.186,148.830
C09870=1149.789,186.262,-61.044,-178.234,7.183,148.830
C09871=1149.794,186.013,-61.020,-178.236,7.181,148.830
C09872=1149.799,185.764,-60.997,-178.239,7.180,148.831
C09873=1149.803,185.515,-60.974,-178.242,7.177,148.831
C09874=1149.808,185.266,-60.950,-178.244,7.175,148.831
C09875=1149.812,185.017,-60.927,-178.248,7.172,148.831
C09876=1149.817,184.769,-60.904,-178.250,7.170,148.832
C09877=1149.822,184.520,-60.881,-178.253,7.168,148.832
C09878=1149.827,184.271,-60.858,-178.256,7.166,148.832
C09879=1149.832,184.001,-60.833,-178.259,7.163,148.832
C09880=1149.837,183.732,-60.808,-178.262,7.161,148.833
C09881=1149.841,183.462,-60.782,-178.265,7.159,148.833
C09882=1149.846,183.192,-60.757,-178.268,7.156,148.833
C09883=1149.851,182.944,-60.735,-178.271,7.153,148.834
C09884=1149.856,182.695,-60.711,-178.273,7.152,148.834
C09885=1149.861,182.445,-60.689,-178.276,7.150,148.834
C09886=1149.865,182.196,-60.665,-178.279,7.147,148.834
C09887=1149.869,181.947,-60.643,-178.282,7.145,148.835
C09888=1149.874,181.698,-60.619,-178.284,7.142,148.835
C09889=1149.879,181.450,-60.596,-178.287,7.141,148.835
C09890=1149.883,181.201,-60.573,-178.290,7.139,148.836
C09891=1149.888,180.952,-60.550,-178.293,7.136,148.836
C09892=1149.893,180.703,-60.527,-178.295,7.134,148.836
C09893=1149.897,180.454,-60.505,-178.298,7.132,148.836
C09894=1149.902,180.206,-60.482,-178.301,7.130,148.837
C09895=1149.906,179.957,-60.459,-178.304,7.127,148.837
C09896=1149.911,179.707,-60.436,-178.307,7.125,148.837
C09897=1149.916,179.458,-60.413,-178.309,7.123,148.837
C09898=1149.920,179.209,-60.390,-178.312,7.121,148.838
C09899=1149.925,178.961,-60.367,-178.315,7.119,148.838
C09900=1149.930,178.712,-60.345,-178.318,7.116,148.838
C09901=1149.934,178.463,-60.322,-178.320,7.114,148.839
C09902=1149.939,178.214,-60.298,-178.323,7.112,148.839
C09903=1149.944,177.965,-60.277,-178.326,7.110,148.839
C09904=1149.949,177.716,-60.253,-178.329,7.108,148.840
C09905=1149.952,177.467,-60.231,-178.332,7.105,148.840
C09906=1149.957,177.218,-60.208,-178.335,7.104,148.840
C09907=1149.962,176.970,-60.186,-178.337,7.101,148.840
C09908=1149.967,176.721,-60.162,-178.340,7.099,148.841
C09909=1149.971,176.471,-60.140,-178.343,7.097,148.841
C09910=1149.976,176.223,-60.117,-178.345,7.095,148.841
C09911=1149.981,175.974,-60.095,-178.348,7.093,148.842
C09912=1149.985,175.725,-60.072,-178.351,7.091,148.842
C09913=1149.989,175.476,-60.049,-178.354,7.088,148.842
C09914=1149.995,175.227,-60.027,-178.356,7.086,148.842
C09915=1149.999,174.978,-60.004,-178.359,7.084,148.843
C09916=1150.004,174.729,-59.981,-178.362,7.082,148.843
C09917=1150.008,174.481,-59.959,-178.365,7.080,148.843
C09918=1150.013,174.231,-59.937,-178.367,7.078,148.844
C09919=1150.017,173.982,-59.913,-178.371,7.075,148.844
C09920=1150.022,173.734,-59.892,-178.373,7.073,148.844
C09921=1150.027,173.484,-59.869,-178.376,7.071,148.844
C09922=1150.031,173.235,-59.846,-178.379,7.069,148.845
C09923=1150.037,172.986,-59.824,-178.382,7.067,148.845
C09924=1150.041,172.737,-59.801,-178.384,7.064,148.845
C09925=1150.045,172.488,-59.779,-178.387,7.063,148.846
C09926=1150.050,172.240,-59.756,-178.390,7.061,148.846
C09927=1150.055,171.990,-59.734,-178.393,7.058,148.846
C09928=1150.059,171.742,-59.713,-178.395,7.056,148.847
C09929=1150.064,171.493,-59.689,-178.398,7.055,148.847
C09930=1150.068,171.243,-59.667,-178.401,7.052,148.847
C09931=1150.073,170.995,-59.645,-178.403,7.050,148.847
C09932=1150.078,170.746,-59.622,-178.406,7.048,148.848
C09933=1150.083,170.497,-59.600,-178.409,7.046,148.848
C09934=1150.087,170.248,-59.578,-178.412,7.044,148.849
C09935=1150.092,169.999,-59.555,-178.414,7.042,148.849
C09936=1150.097,169.750,-59.533,-178.418,7.039,148.849
C09937=1150.101,169.501,-59.511,-178.420,7.038,148.849
C09938=1150.107,169.252,-59.489,-178.423,7.036,148.850
C09939=1150.111,169.003,-59.466,-178.426,7.033,148.850
C09940=1150.115,168.754,-59.445,-178.429,7.031,148.850
C09941=1150.120,168.505,-59.423,-178.431,7.029,148.851
C09942=1150.125,168.256,-59.400,-178.434,7.027,148.851
C09943=1150.130,168.007,-59.378,-178.437,7.025,148.851
C09944=1150.134,167.759,-59.356,-178.439,7.023,148.852
C09945=1150.138,167.509,-59.334,-178.443,7.021,148.852
C09946=1150.143,167.260,-59.311,-178.445,7.019,148.852
C09947=1150.148,167.011,-59.289,-178.448,7.017,148.853
C09948=1150.153,166.762,-59.267,-178.451,7.014,148.853
C09949=1150.157,166.513,-59.246,-178.454,7.012,148.853
C09950=1150.162,166.264,-59.224,-178.456,7.011,148.854
C09951=1150.167,166.016,-59.201,-178.459,7.009,148.854
C09952=1150.171,165.766,-59.179,-178.462,7.006,148.854
C09953=1150.176,165.518,-59.157,-178.465,7.004,148.854
C09954=1150.180,165.268,-59.135,-178.467,7.003,148.855
C09955=1150.185,165.020,-59.113,-178.471,7.000,148.855
C09956=1150.190,164.771,-59.092,-178.473,6.998,148.855
C09957=1150.194,164.522,-59.069,-178.475,6.996,148.856
C09958=1150.200,164.273,-59.047,-178.479,6.994,148.856
C09959=1150.204,164.023,-59.025,-178.481,6.992,148.856
C09960=1150.209,163.775,-59.003,-178.484,6.990,148.857
C09961=1150.213,163.525,-58.981,-178.487,6.989,148.857
C09962=1150.218,163.277,-58.960,-178.490,6.986,148.857
C09963=1150.223,163.027,-58.938,-178.492,6.984,148.858
C09964=1150.227,162.779,-58.916,-178.495,6.982,148.858
C09965=1150.232,162.529,-58.894,-178.498,6.980,148.858
C09966=1150.237,162.281,-58.872,-178.501,6.978,148.859
C09967=1150.241,162.032,-58.851,-178.503,6.976,148.859
C09968=1150.246,161.783,-58.829,-178.506,6.974,148.859
C09969=1150.251,161.533,-58.808,-178.509,6.972,148.860
C09970=1150.255,161.284,-58.786,-178.512,6.970,148.860
C09971=1150.260,161.035,-58.764,-178.515,6.968,148.860
C09972=1150.265,160.787,-58.742,-178.517,6.966,148.861
C09973=1150.269,160.538,-58.720,-178.520,6.963,148.861
C09974=1150.274,160.289,-58.698,-178.523,6.962,148.861
C09975=1150.279,160.039,-58.677,-178.526,6.960,148.862
C09976=1150.283,159.790,-58.655,-178.528,6.958,148.862
C09977=1150.288,159.542,-58.634,-178.532,6.956,148.862
C09978=1150.293,159.292,-58.612,-178.534,6.954,148.863
C09979=1150.297,159.044,-58.590,-178.536,6.952,148.863
C09980=1150.303,158.794,-58.569,-178.539,6.950,148.863
C09981=1150.307,158.545,-58.547,-178.542,6.948,148.864
C09982=1150.312,158.296,-58.525,-178.545,6.946,148.864
C09983=1150.316,158.027,-58.503,-178.548,6.944,148.864
C09984=1150.322,157.758,-58.479,-178.551,6.942,148.865
C09985=1150.327,157.489,-58.455,-178.554,6.940,148.865
C09986=1150.332,157.220,-58.432,-178.557,6.937,148.865
C09987=1150.337,156.972,-58.411,-178.560,6.936,148.866
C09988=1150.342,156.722,-58.390,-178.563,6.934,148.866
C09989=1150.346,156.473,-58.368,-178.565,6.931,148.866
C09990=1150.351,156.224,-58.346,-178.568,6.929,148.867
C09991=1150.356,155.975,-58.326,-178.571,6.928,148.867
C09992=1150.360,155.726,-58.304,-178.573,6.926,148.868
C09993=1150.365,155.477,-58.282,-178.576,6.924,148.868
C09994=1150.370,155.228,-58.261,-178.579,6.922,148.868
C09995=1150.374,154.979,-58.239,-178.582,6.920,148.869
C09996=1150.379,154.730,-58.218,-178.584,6.918,148.869
//INST
///DATE 2021/06/15 17:27
///ATTR SC,RW,RJ
////FRAME ROBOT
///GROUP1 RB1
NOP
MOVL C00000 V=800.0 PL=0
MOVL C00001 V=800.0 PL=0
MOVL C00002 V=800.0 PL=0
MOVL C00003 V=800.0 PL=0
MOVL C00004 V=800.0 PL=0
MOVL C00005 V=800.0 PL=0
MOVL C00006 V=800.0 PL=0
MOVL C00007 V=800.0 PL=0
MOVL C00008 V=800.0 PL=0
MOVL C00009 V=800.0 PL=0
MOVL C00010 V=800.0 PL=0
MOVL C00011 V=800.0 PL=0
MOVL C00012 V=800.0 PL=0
MOVL C00013 V=800.0 PL=0
MOVL C00014 V=800.0 PL=0
MOVL C00015 V=800.0 PL=0
MOVL C00016 V=800.0 PL=0
MOVL C00017 V=800.0 PL=0
MOVL C00018 V=800.0 PL=0
MOVL C00019 V=800.0 PL=0
MOVL C00020 V=800.0 PL=0
MOVL C00021 V=800.0 PL=0
MOVL C00022 V=800.0 PL=0
MOVL C00023 V=800.0 PL=0
MOVL C00024 V=800.0 PL=0
MOVL C00025 V=800.0 PL=0
MOVL C00026 V=800.0 PL=0
MOVL C00027 V=800.0 PL=0
MOVL C00028 V=800.0 PL=0
MOVL C00029 V=800.0 PL=0
MOVL C00030 V=800.0 PL=0
MOVL C00031 V=800.0 PL=0
MOVL C00032 V=800.0 PL=0
MOVL C00033 V=800.0 PL=0
MOVL C00034 V=800.0 PL=0
MOVL C00035 V=800.0 PL=0
MOVL C00036 V=800.0 PL=0
MOVL C00037 V=800.0 PL=0
MOVL C00038 V=800.0 PL=0
MOVL C00039 V=800.0 PL=0
MOVL C00040 V=800.0 PL=0
MOVL C00041 V=800.0 PL=0
MOVL C00042 V=800.0 PL=0
MOVL C00043 V=800.0 PL=0
MOVL C00044 V=800.0 PL=0
MOVL C00045 V=800.0 PL=0
MOVL C00046 V=800.0 PL=0
MOVL C00047 V=800.0 PL=0
MOVL C00048 V=800.0 PL=0
MOVL C00049 V=800.0 PL=0
MOVL C00050 V=800.0 PL=0
MOVL C00051 V=800.0 PL=0
MOVL C00052 V=800.0 PL=0
MOVL C00053 V=800.0 PL=0
MOVL C00054 V=800.0 PL=0
MOVL C00055 V=800.0 PL=0
MOVL C00056 V=800.0 PL=0
MOVL C00057 V=800.0 PL=0
MOVL C00058 V=800.0 PL=0
MOVL C00059 V=800.0 PL=0
MOVL C00060 V=800.0 PL=0
MOVL C00061 V=800.0 PL=0
MOVL C00062 V=800.0 PL=0
MOVL C00063 V=800.0 PL=0
MOVL C00064 V=800.0 PL=0
MOVL C00065 V=800.0 PL=0
MOVL C00066 V=800.0 PL=0
MOVL C00067 V=800.0 PL=0
MOVL C00068 V=800.0 PL=0
MOVL C00069 V=800.0 PL=0
MOVL C00070 V=800.0 PL=0
MOVL C00071 V=800.0 PL=0
MOVL C00072 V=800.0 PL=0
MOVL C00073 V=800.0 PL=0
MOVL C00074 V=800.0 PL=0
MOVL C00075 V=800.0 PL=0
MOVL C00076 V=800.0 PL=0
MOVL C00077 V=800.0 PL=0
MOVL C00078 V=800.0 PL=0
MOVL C00079 V=800.0 PL=0
MOVL C00080 V=800.0 PL=0
MOVL C00081 V=800.0 PL=0
MOVL C00082 V=800.0 PL=0
MOVL C00083 V=800.0 PL=0
MOVL C00084 V=800.0 PL=0
MOVL C00085 V=800.0 PL=0
MOVL C00086 V=800.0 PL=0
MOVL C00087 V=800.0 PL=0
MOVL C00088 V=800.0 PL=0
MOVL C00089 V=800.0 PL=0
MOVL C00090 V=800.0 PL=0
MOVL C00091 V=800.0 PL=0
MOVL C00092 V=800.0 PL=0
MOVL C00093 V=800.0 PL=0
MOVL C00094 V=800.0 PL=0
MOVL C00095 V=800.0 PL=0
MOVL C00096 V=800.0 PL=0
MOVL C00097 V=800.0 PL=0
MOVL C00098 V=800.0 PL=0
MOVL C00099 V=800.0 PL=0
MOVL C00100 V=800.0 PL=0
MOVL C00101 V=800.0 PL=0
MOVL C00102 V=800.0 PL=0
MOVL C00103 V=800.0 PL=0
MOVL C00104 V=800.0 PL=0
MOVL C00105 V=800.0 PL=0
MOVL C00106 V=800.0 PL=0
MOVL C00107 V=800.0 PL=0
MOVL C00108 V=800.0 PL=0
MOVL C00109 V=800.0 PL=0
MOVL C00110 V=800.0 PL=0
MOVL C00111 V=800.0 PL=0
MOVL C00112 V=800.0 PL=0
MOVL C00113 V=800.0 PL=0
MOVL C00114 V=800.0 PL=0
MOVL C00115 V=800.0 PL=0
MOVL C00116 V=800.0 PL=0
MOVL C00117 V=800.0 PL=0
MOVL C00118 V=800.0 PL=0
MOVL C00119 V=800.0 PL=0
MOVL C00120 V=800.0 PL=0
MOVL C00121 V=800.0 PL=0
MOVL C00122 V=800.0 PL=0
MOVL C00123 V=800.0 PL=0
MOVL C00124 V=800.0 PL=0
MOVL C00125 V=800.0 PL=0
MOVL C00126 V=800.0 PL=0
MOVL C00127 V=800.0 PL=0
MOVL C00128 V=800.0 PL=0
MOVL C00129 V=800.0 PL=0
MOVL C00130 V=800.0 PL=0
MOVL C00131 V=800.0 PL=0
MOVL C00132 V=800.0 PL=0
MOVL C00133 V=800.0 PL=0
MOVL C00134 V=800.0 PL=0
MOVL C00135 V=800.0 PL=0
MOVL C00136 V=800.0 PL=0
MOVL C00137 V=800.0 PL=0
MOVL C00138 V=800.0 PL=0
MOVL C00139 V=800.0 PL=0
MOVL C00140 V=800.0 PL=0
MOVL C00141 V=800.0 PL=0
MOVL C00142 V=800.0 PL=0
MOVL C00143 V=800.0 PL=0
MOVL C00144 V=800.0 PL=0
MOVL C00145 V=800.0 PL=0
MOVL C00146 V=800.0 PL=0
MOVL C00147 V=800.0 PL=0
MOVL C00148 V=800.0 PL=0
MOVL C00149 V=800.0 PL=0
MOVL C00150 V=800.0 PL=0
MOVL C00151 V=800.0 PL=0
MOVL C00152 V=800.0 PL=0
MOVL C00153 V=800.0 PL=0
MOVL C00154 V=800.0 PL=0
MOVL C00155 V=800.0 PL=0
MOVL C00156 V=800.0 PL=0
MOVL C00157 V=800.0 PL=0
MOVL C00158 V=800.0 PL=0
MOVL C00159 V=800.0 PL=0
MOVL C00160 V=800.0 PL=0
MOVL C00161 V=800.0 PL=0
MOVL C00162 V=800.0 PL=0
MOVL C00163 V=800.0 PL=0
MOVL C00164 V=800.0 PL=0
MOVL C00165 V=800.0 PL=0
MOVL C00166 V=800.0 PL=0
MOVL C00167 V=800.0 PL=0
MOVL C00168 V=800.0 PL=0
MOVL C00169 V=800.0 PL=0
MOVL C00170 V=800.0 PL=0
MOVL C00171 V=800.0 PL=0
MOVL C00172 V=800.0 PL=0
MOVL C00173 V=800.0 PL=0
MOVL C00174 V=800.0 PL=0
MOVL C00175 V=800.0 PL=0
MOVL C00176 V=800.0 PL=0
MOVL C00177 V=800.0 PL=0
MOVL C00178 V=800.0 PL=0
MOVL C00179 V=800.0 PL=0
MOVL C00180 V=800.0 PL=0
MOVL C00181 V=800.0 PL=0
MOVL C00182 V=800.0 PL=0
MOVL C00183 V=800.0 PL=0
MOVL C00184 V=800.0 PL=0
MOVL C00185 V=800.0 PL=0
MOVL C00186 V=800.0 PL=0
MOVL C00187 V=800.0 PL=0
MOVL C00188 V=800.0 PL=0
MOVL C00189 V=800.0 PL=0
MOVL C00190 V=800.0 PL=0
MOVL C00191 V=800.0 PL=0
MOVL C00192 V=800.0 PL=0
MOVL C00193 V=800.0 PL=0
MOVL C00194 V=800.0 PL=0
MOVL C00195 V=800.0 PL=0
MOVL C00196 V=800.0 PL=0
MOVL C00197 V=800.0 PL=0
MOVL C00198 V=800.0 PL=0
MOVL C00199 V=800.0 PL=0
MOVL C00200 V=800.0 PL=0
MOVL C00201 V=800.0 PL=0
MOVL C00202 V=800.0 PL=0
MOVL C00203 V=800.0 PL=0
MOVL C00204 V=800.0 PL=0
MOVL C00205 V=800.0 PL=0
MOVL C00206 V=800.0 PL=0
MOVL C00207 V=800.0 PL=0
MOVL C00208 V=800.0 PL=0
MOVL C00209 V=800.0 PL=0
MOVL C00210 V=800.0 PL=0
MOVL C00211 V=800.0 PL=0
MOVL C00212 V=800.0 PL=0
MOVL C00213 V=800.0 PL=0
MOVL C00214 V=800.0 PL=0
MOVL C00215 V=800.0 PL=0
MOVL C00216 V=800.0 PL=0
MOVL C00217 V=800.0 PL=0
MOVL C00218 V=800.0 PL=0
MOVL C00219 V=800.0 PL=0
MOVL C00220 V=800.0 PL=0
MOVL C00221 V=800.0 PL=0
MOVL C00222 V=800.0 PL=0
MOVL C00223 V=800.0 PL=0
MOVL C00224 V=800.0 PL=0
MOVL C00225 V=800.0 PL=0
MOVL C00226 V=800.0 PL=0
MOVL C00227 V=800.0 PL=0
MOVL C00228 V=800.0 PL=0
MOVL C00229 V=800.0 PL=0
MOVL C00230 V=800.0 PL=0
MOVL C00231 V=800.0 PL=0
MOVL C00232 V=800.0 PL=0
MOVL C00233 V=800.0 PL=0
MOVL C00234 V=800.0 PL=0
MOVL C00235 V=800.0 PL=0
MOVL C00236 V=800.0 PL=0
MOVL C00237 V=800.0 PL=0
MOVL C00238 V=800.0 PL=0
MOVL C00239 V=800.0 PL=0
MOVL C00240 V=800.0 PL=0
MOVL C00241 V=800.0 PL=0
MOVL C00242 V=800.0 PL=0
MOVL C00243 V=800.0 PL=0
MOVL C00244 V=800.0 PL=0
MOVL C00245 V=800.0 PL=0
MOVL C00246 V=800.0 PL=0
MOVL C00247 V=800.0 PL=0
MOVL C00248 V=800.0 PL=0
MOVL C00249 V=800.0 PL=0
MOVL C00250 V=800.0 PL=0
MOVL C00251 V=800.0 PL=0
MOVL C00252 V=800.0 PL=0
MOVL C00253 V=800.0 PL=0
MOVL C00254 V=800.0 PL=0
MOVL C00255 V=800.0 PL=0
MOVL C00256 V=800.0 PL=0
MOVL C00257 V=800.0 PL=0
MOVL C00258 V=800.0 PL=0
MOVL C00259 V=800.0 PL=0
MOVL C00260 V=800.0 PL=0
MOVL C00261 V=800.0 PL=0
MOVL C00262 V=800.0 PL=0
MOVL C00263 V=800.0 PL=0
MOVL C00264 V=800.0 PL=0
MOVL C00265 V=800.0 PL=0
MOVL C00266 V=800.0 PL=0
MOVL C00267 V=800.0 PL=0
MOVL C00268 V=800.0 PL=0
MOVL C00269 V=800.0 PL=0
MOVL C00270 V=800.0 PL=0
MOVL C00271 V=800.0 PL=0
MOVL C00272 V=800.0 PL=0
MOVL C00273 V=800.0 PL=0
MOVL C00274 V=800.0 PL=0
MOVL C00275 V=800.0 PL=0
MOVL C00276 V=800.0 PL=0
MOVL C00277 V=800.0 PL=0
MOVL C00278 V=800.0 PL=0
MOVL C00279 V=800.0 PL=0
MOVL C00280 V=800.0 PL=0
MOVL C00281 V=800.0 PL=0
MOVL C00282 V=800.0 PL=0
MOVL C00283 V=800.0 PL=0
MOVL C00284 V=800.0 PL=0
MOVL C00285 V=800.0 PL=0
MOVL C00286 V=800.0 PL=0
MOVL C00287 V=800.0 PL=0
MOVL C00288 V=800.0 PL=0
MOVL C00289 V=800.0 PL=0
MOVL C00290 V=800.0 PL=0
MOVL C00291 V=800.0 PL=0
MOVL C00292 V=800.0 PL=0
MOVL C00293 V=800.0 PL=0
MOVL C00294 V=800.0 PL=0
MOVL C00295 V=800.0 PL=0
MOVL C00296 V=800.0 PL=0
MOVL C00297 V=800.0 PL=0
MOVL C00298 V=800.0 PL=0
MOVL C00299 V=800.0 PL=0
MOVL C00300 V=800.0 PL=0
MOVL C00301 V=800.0 PL=0
MOVL C00302 V=800.0 PL=0
MOVL C00303 V=800.0 PL=0
MOVL C00304 V=800.0 PL=0
MOVL C00305 V=800.0 PL=0
MOVL C00306 V=800.0 PL=0
MOVL C00307 V=800.0 PL=0
MOVL C00308 V=800.0 PL=0
MOVL C00309 V=800.0 PL=0
MOVL C00310 V=800.0 PL=0
MOVL C00311 V=800.0 PL=0
MOVL C00312 V=800.0 PL=0
MOVL C00313 V=800.0 PL=0
MOVL C00314 V=800.0 PL=0
MOVL C00315 V=800.0 PL=0
MOVL C00316 V=800.0 PL=0
MOVL C00317 V=800.0 PL=0
MOVL C00318 V=800.0 PL=0
MOVL C00319 V=800.0 PL=0
MOVL C00320 V=800.0 PL=0
MOVL C00321 V=800.0 PL=0
MOVL C00322 V=800.0 PL=0
MOVL C00323 V=800.0 PL=0
MOVL C00324 V=800.0 PL=0
MOVL C00325 V=800.0 PL=0
MOVL C00326 V=800.0 PL=0
MOVL C00327 V=800.0 PL=0
MOVL C00328 V=800.0 PL=0
MOVL C00329 V=800.0 PL=0
MOVL C00330 V=800.0 PL=0
MOVL C00331 V=800.0 PL=0
MOVL C00332 V=800.0 PL=0
MOVL C00333 V=800.0 PL=0
MOVL C00334 V=800.0 PL=0
MOVL C00335 V=800.0 PL=0
MOVL C00336 V=800.0 PL=0
MOVL C00337 V=800.0 PL=0
MOVL C00338 V=800.0 PL=0
MOVL C00339 V=800.0 PL=0
MOVL C00340 V=800.0 PL=0
MOVL C00341 V=800.0 PL=0
MOVL C00342 V=800.0 PL=0
MOVL C00343 V=800.0 PL=0
MOVL C00344 V=800.0 PL=0
MOVL C00345 V=800.0 PL=0
MOVL C00346 V=800.0 PL=0
MOVL C00347 V=800.0 PL=0
MOVL C00348 V=800.0 PL=0
MOVL C00349 V=800.0 PL=0
MOVL C00350 V=800.0 PL=0
MOVL C00351 V=800.0 PL=0
MOVL C00352 V=800.0 PL=0
MOVL C00353 V=800.0 PL=0
MOVL C00354 V=800.0 PL=0
MOVL C00355 V=800.0 PL=0
MOVL C00356 V=800.0 PL=0
MOVL C00357 V=800.0 PL=0
MOVL C00358 V=800.0 PL=0
MOVL C00359 V=800.0 PL=0
MOVL C00360 V=800.0 PL=0
MOVL C00361 V=800.0 PL=0
MOVL C00362 V=800.0 PL=0
MOVL C00363 V=800.0 PL=0
MOVL C00364 V=800.0 PL=0
MOVL C00365 V=800.0 PL=0
MOVL C00366 V=800.0 PL=0
MOVL C00367 V=800.0 PL=0
MOVL C00368 V=800.0 PL=0
MOVL C00369 V=800.0 PL=0
MOVL C00370 V=800.0 PL=0
MOVL C00371 V=800.0 PL=0
MOVL C00372 V=800.0 PL=0
MOVL C00373 V=800.0 PL=0
MOVL C00374 V=800.0 PL=0
MOVL C00375 V=800.0 PL=0
MOVL C00376 V=800.0 PL=0
MOVL C00377 V=800.0 PL=0
MOVL C00378 V=800.0 PL=0
MOVL C00379 V=800.0 PL=0
MOVL C00380 V=800.0 PL=0
MOVL C00381 V=800.0 PL=0
MOVL C00382 V=800.0 PL=0
MOVL C00383 V=800.0 PL=0
MOVL C00384 V=800.0 PL=0
MOVL C00385 V=800.0 PL=0
MOVL C00386 V=800.0 PL=0
MOVL C00387 V=800.0 PL=0
MOVL C00388 V=800.0 PL=0
MOVL C00389 V=800.0 PL=0
MOVL C00390 V=800.0 PL=0
MOVL C00391 V=800.0 PL=0
MOVL C00392 V=800.0 PL=0
MOVL C00393 V=800.0 PL=0
MOVL C00394 V=800.0 PL=0
MOVL C00395 V=800.0 PL=0
MOVL C00396 V=800.0 PL=0
MOVL C00397 V=800.0 PL=0
MOVL C00398 V=800.0 PL=0
MOVL C00399 V=800.0 PL=0
MOVL C00400 V=800.0 PL=0
MOVL C00401 V=800.0 PL=0
MOVL C00402 V=800.0 PL=0
MOVL C00403 V=800.0 PL=0
MOVL C00404 V=800.0 PL=0
MOVL C00405 V=800.0 PL=0
MOVL C00406 V=800.0 PL=0
MOVL C00407 V=800.0 PL=0
MOVL C00408 V=800.0 PL=0
MOVL C00409 V=800.0 PL=0
MOVL C00410 V=800.0 PL=0
MOVL C00411 V=800.0 PL=0
MOVL C00412 V=800.0 PL=0
MOVL C00413 V=800.0 PL=0
MOVL C00414 V=800.0 PL=0
MOVL C00415 V=800.0 PL=0
MOVL C00416 V=800.0 PL=0
MOVL C00417 V=800.0 PL=0
MOVL C00418 V=800.0 PL=0
MOVL C00419 V=800.0 PL=0
MOVL C00420 V=800.0 PL=0
MOVL C00421 V=800.0 PL=0
MOVL C00422 V=800.0 PL=0
MOVL C00423 V=800.0 PL=0
MOVL C00424 V=800.0 PL=0
MOVL C00425 V=800.0 PL=0
MOVL C00426 V=800.0 PL=0
MOVL C00427 V=800.0 PL=0
MOVL C00428 V=800.0 PL=0
MOVL C00429 V=800.0 PL=0
MOVL C00430 V=800.0 PL=0
MOVL C00431 V=800.0 PL=0
MOVL C00432 V=800.0 PL=0
MOVL C00433 V=800.0 PL=0
MOVL C00434 V=800.0 PL=0
MOVL C00435 V=800.0 PL=0
MOVL C00436 V=800.0 PL=0
MOVL C00437 V=800.0 PL=0
MOVL C00438 V=800.0 PL=0
MOVL C00439 V=800.0 PL=0
MOVL C00440 V=800.0 PL=0
MOVL C00441 V=800.0 PL=0
MOVL C00442 V=800.0 PL=0
MOVL C00443 V=800.0 PL=0
MOVL C00444 V=800.0 PL=0
MOVL C00445 V=800.0 PL=0
MOVL C00446 V=800.0 PL=0
MOVL C00447 V=800.0 PL=0
MOVL C00448 V=800.0 PL=0
MOVL C00449 V=800.0 PL=0
MOVL C00450 V=800.0 PL=0
MOVL C00451 V=800.0 PL=0
MOVL C00452 V=800.0 PL=0
MOVL C00453 V=800.0 PL=0
MOVL C00454 V=800.0 PL=0
MOVL C00455 V=800.0 PL=0
MOVL C00456 V=800.0 PL=0
MOVL C00457 V=800.0 PL=0
MOVL C00458 V=800.0 PL=0
MOVL C00459 V=800.0 PL=0
MOVL C00460 V=800.0 PL=0
MOVL C00461 V=800.0 PL=0
MOVL C00462 V=800.0 PL=0
MOVL C00463 V=800.0 PL=0
MOVL C00464 V=800.0 PL=0
MOVL C00465 V=800.0 PL=0
MOVL C00466 V=800.0 PL=0
MOVL C00467 V=800.0 PL=0
MOVL C00468 V=800.0 PL=0
MOVL C00469 V=800.0 PL=0
MOVL C00470 V=800.0 PL=0
MOVL C00471 V=800.0 PL=0
MOVL C00472 V=800.0 PL=0
MOVL C00473 V=800.0 PL=0
MOVL C00474 V=800.0 PL=0
MOVL C00475 V=800.0 PL=0
MOVL C00476 V=800.0 PL=0
MOVL C00477 V=800.0 PL=0
MOVL C00478 V=800.0 PL=0
MOVL C00479 V=800.0 PL=0
MOVL C00480 V=800.0 PL=0
MOVL C00481 V=800.0 PL=0
MOVL C00482 V=800.0 PL=0
MOVL C00483 V=800.0 PL=0
MOVL C00484 V=800.0 PL=0
MOVL C00485 V=800.0 PL=0
MOVL C00486 V=800.0 PL=0
MOVL C00487 V=800.0 PL=0
MOVL C00488 V=800.0 PL=0
MOVL C00489 V=800.0 PL=0
MOVL C00490 V=800.0 PL=0
MOVL C00491 V=800.0 PL=0
MOVL C00492 V=800.0 PL=0
MOVL C00493 V=800.0 PL=0
MOVL C00494 V=800.0 PL=0
MOVL C00495 V=800.0 PL=0
MOVL C00496 V=800.0 PL=0
MOVL C00497 V=800.0 PL=0
MOVL C00498 V=800.0 PL=0
MOVL C00499 V=800.0 PL=0
MOVL C00500 V=800.0 PL=0
MOVL C00501 V=800.0 PL=0
MOVL C00502 V=800.0 PL=0
MOVL C00503 V=800.0 PL=0
MOVL C00504 V=800.0 PL=0
MOVL C00505 V=800.0 PL=0
MOVL C00506 V=800.0 PL=0
MOVL C00507 V=800.0 PL=0
MOVL C00508 V=800.0 PL=0
MOVL C00509 V=800.0 PL=0
MOVL C00510 V=800.0 PL=0
MOVL C00511 V=800.0 PL=0
MOVL C00512 V=800.0 PL=0
MOVL C00513 V=800.0 PL=0
MOVL C00514 V=800.0 PL=0
MOVL C00515 V=800.0 PL=0
MOVL C00516 V=800.0 PL=0
MOVL C00517 V=800.0 PL=0
MOVL C00518 V=800.0 PL=0
MOVL C00519 V=800.0 PL=0
MOVL C00520 V=800.0 PL=0
MOVL C00521 V=800.0 PL=0
MOVL C00522 V=800.0 PL=0
MOVL C00523 V=800.0 PL=0
MOVL C00524 V=800.0 PL=0
MOVL C00525 V=800.0 PL=0
MOVL C00526 V=800.0 PL=0
MOVL C00527 V=800.0 PL=0
MOVL C00528 V=800.0 PL=0
MOVL C00529 V=800.0 PL=0
MOVL C00530 V=800.0 PL=0
MOVL C00531 V=800.0 PL=0
MOVL C00532 V=800.0 PL=0
MOVL C00533 V=800.0 PL=0
MOVL C00534 V=800.0 PL=0
MOVL C00535 V=800.0 PL=0
MOVL C00536 V=800.0 PL=0
MOVL C00537 V=800.0 PL=0
MOVL C00538 V=800.0 PL=0
MOVL C00539 V=800.0 PL=0
MOVL C00540 V=800.0 PL=0
MOVL C00541 V=800.0 PL=0
MOVL C00542 V=800.0 PL=0
MOVL C00543 V=800.0 PL=0
MOVL C00544 V=800.0 PL=0
MOVL C00545 V=800.0 PL=0
MOVL C00546 V=800.0 PL=0
MOVL C00547 V=800.0 PL=0
MOVL C00548 V=800.0 PL=0
MOVL C00549 V=800.0 PL=0
MOVL C00550 V=800.0 PL=0
MOVL C00551 V=800.0 PL=0
MOVL C00552 V=800.0 PL=0
MOVL C00553 V=800.0 PL=0
MOVL C00554 V=800.0 PL=0
MOVL C00555 V=800.0 PL=0
MOVL C00556 V=800.0 PL=0
MOVL C00557 V=800.0 PL=0
MOVL C00558 V=800.0 PL=0
MOVL C00559 V=800.0 PL=0
MOVL C00560 V=800.0 PL=0
MOVL C00561 V=800.0 PL=0
MOVL C00562 V=800.0 PL=0
MOVL C00563 V=800.0 PL=0
MOVL C00564 V=800.0 PL=0
MOVL C00565 V=800.0 PL=0
MOVL C00566 V=800.0 PL=0
MOVL C00567 V=800.0 PL=0
MOVL C00568 V=800.0 PL=0
MOVL C00569 V=800.0 PL=0
MOVL C00570 V=800.0 PL=0
MOVL C00571 V=800.0 PL=0
MOVL C00572 V=800.0 PL=0
MOVL C00573 V=800.0 PL=0
MOVL C00574 V=800.0 PL=0
MOVL C00575 V=800.0 PL=0
MOVL C00576 V=800.0 PL=0
MOVL C00577 V=800.0 PL=0
MOVL C00578 V=800.0 PL=0
MOVL C00579 V=800.0 PL=0
MOVL C00580 V=800.0 PL=0
MOVL C00581 V=800.0 PL=0
MOVL C00582 V=800.0 PL=0
MOVL C00583 V=800.0 PL=0
MOVL C00584 V=800.0 PL=0
MOVL C00585 V=800.0 PL=0
MOVL C00586 V=800.0 PL=0
MOVL C00587 V=800.0 PL=0
MOVL C00588 V=800.0 PL=0
MOVL C00589 V=800.0 PL=0
MOVL C00590 V=800.0 PL=0
MOVL C00591 V=800.0 PL=0
MOVL C00592 V=800.0 PL=0
MOVL C00593 V=800.0 PL=0
MOVL C00594 V=800.0 PL=0
MOVL C00595 V=800.0 PL=0
MOVL C00596 V=800.0 PL=0
MOVL C00597 V=800.0 PL=0
MOVL C00598 V=800.0 PL=0
MOVL C00599 V=800.0 PL=0
MOVL C00600 V=800.0 PL=0
MOVL C00601 V=800.0 PL=0
MOVL C00602 V=800.0 PL=0
MOVL C00603 V=800.0 PL=0
MOVL C00604 V=800.0 PL=0
MOVL C00605 V=800.0 PL=0
MOVL C00606 V=800.0 PL=0
MOVL C00607 V=800.0 PL=0
MOVL C00608 V=800.0 PL=0
MOVL C00609 V=800.0 PL=0
MOVL C00610 V=800.0 PL=0
MOVL C00611 V=800.0 PL=0
MOVL C00612 V=800.0 PL=0
MOVL C00613 V=800.0 PL=0
MOVL C00614 V=800.0 PL=0
MOVL C00615 V=800.0 PL=0
MOVL C00616 V=800.0 PL=0
MOVL C00617 V=800.0 PL=0
MOVL C00618 V=800.0 PL=0
MOVL C00619 V=800.0 PL=0
MOVL C00620 V=800.0 PL=0
MOVL C00621 V=800.0 PL=0
MOVL C00622 V=800.0 PL=0
MOVL C00623 V=800.0 PL=0
MOVL C00624 V=800.0 PL=0
MOVL C00625 V=800.0 PL=0
MOVL C00626 V=800.0 PL=0
MOVL C00627 V=800.0 PL=0
MOVL C00628 V=800.0 PL=0
MOVL C00629 V=800.0 PL=0
MOVL C00630 V=800.0 PL=0
MOVL C00631 V=800.0 PL=0
MOVL C00632 V=800.0 PL=0
MOVL C00633 V=800.0 PL=0
MOVL C00634 V=800.0 PL=0
MOVL C00635 V=800.0 PL=0
MOVL C00636 V=800.0 PL=0
MOVL C00637 V=800.0 PL=0
MOVL C00638 V=800.0 PL=0
MOVL C00639 V=800.0 PL=0
MOVL C00640 V=800.0 PL=0
MOVL C00641 V=800.0 PL=0
MOVL C00642 V=800.0 PL=0
MOVL C00643 V=800.0 PL=0
MOVL C00644 V=800.0 PL=0
MOVL C00645 V=800.0 PL=0
MOVL C00646 V=800.0 PL=0
MOVL C00647 V=800.0 PL=0
MOVL C00648 V=800.0 PL=0
MOVL C00649 V=800.0 PL=0
MOVL C00650 V=800.0 PL=0
MOVL C00651 V=800.0 PL=0
MOVL C00652 V=800.0 PL=0
MOVL C00653 V=800.0 PL=0
MOVL C00654 V=800.0 PL=0
MOVL C00655 V=800.0 PL=0
MOVL C00656 V=800.0 PL=0
MOVL C00657 V=800.0 PL=0
MOVL C00658 V=800.0 PL=0
MOVL C00659 V=800.0 PL=0
MOVL C00660 V=800.0 PL=0
MOVL C00661 V=800.0 PL=0
MOVL C00662 V=800.0 PL=0
MOVL C00663 V=800.0 PL=0
MOVL C00664 V=800.0 PL=0
MOVL C00665 V=800.0 PL=0
MOVL C00666 V=800.0 PL=0
MOVL C00667 V=800.0 PL=0
MOVL C00668 V=800.0 PL=0
MOVL C00669 V=800.0 PL=0
MOVL C00670 V=800.0 PL=0
MOVL C00671 V=800.0 PL=0
MOVL C00672 V=800.0 PL=0
MOVL C00673 V=800.0 PL=0
MOVL C00674 V=800.0 PL=0
MOVL C00675 V=800.0 PL=0
MOVL C00676 V=800.0 PL=0
MOVL C00677 V=800.0 PL=0
MOVL C00678 V=800.0 PL=0
MOVL C00679 V=800.0 PL=0
MOVL C00680 V=800.0 PL=0
MOVL C00681 V=800.0 PL=0
MOVL C00682 V=800.0 PL=0
MOVL C00683 V=800.0 PL=0
MOVL C00684 V=800.0 PL=0
MOVL C00685 V=800.0 PL=0
MOVL C00686 V=800.0 PL=0
MOVL C00687 V=800.0 PL=0
MOVL C00688 V=800.0 PL=0
MOVL C00689 V=800.0 PL=0
MOVL C00690 V=800.0 PL=0
MOVL C00691 V=800.0 PL=0
MOVL C00692 V=800.0 PL=0
MOVL C00693 V=800.0 PL=0
MOVL C00694 V=800.0 PL=0
MOVL C00695 V=800.0 PL=0
MOVL C00696 V=800.0 PL=0
MOVL C00697 V=800.0 PL=0
MOVL C00698 V=800.0 PL=0
MOVL C00699 V=800.0 PL=0
MOVL C00700 V=800.0 PL=0
MOVL C00701 V=800.0 PL=0
MOVL C00702 V=800.0 PL=0
MOVL C00703 V=800.0 PL=0
MOVL C00704 V=800.0 PL=0
MOVL C00705 V=800.0 PL=0
MOVL C00706 V=800.0 PL=0
MOVL C00707 V=800.0 PL=0
MOVL C00708 V=800.0 PL=0
MOVL C00709 V=800.0 PL=0
MOVL C00710 V=800.0 PL=0
MOVL C00711 V=800.0 PL=0
MOVL C00712 V=800.0 PL=0
MOVL C00713 V=800.0 PL=0
MOVL C00714 V=800.0 PL=0
MOVL C00715 V=800.0 PL=0
MOVL C00716 V=800.0 PL=0
MOVL C00717 V=800.0 PL=0
MOVL C00718 V=800.0 PL=0
MOVL C00719 V=800.0 PL=0
MOVL C00720 V=800.0 PL=0
MOVL C00721 V=800.0 PL=0
MOVL C00722 V=800.0 PL=0
MOVL C00723 V=800.0 PL=0
MOVL C00724 V=800.0 PL=0
MOVL C00725 V=800.0 PL=0
MOVL C00726 V=800.0 PL=0
MOVL C00727 V=800.0 PL=0
MOVL C00728 V=800.0 PL=0
MOVL C00729 V=800.0 PL=0
MOVL C00730 V=800.0 PL=0
MOVL C00731 V=800.0 PL=0
MOVL C00732 V=800.0 PL=0
MOVL C00733 V=800.0 PL=0
MOVL C00734 V=800.0 PL=0
MOVL C00735 V=800.0 PL=0
MOVL C00736 V=800.0 PL=0
MOVL C00737 V=800.0 PL=0
MOVL C00738 V=800.0 PL=0
MOVL C00739 V=800.0 PL=0
MOVL C00740 V=800.0 PL=0
MOVL C00741 V=800.0 PL=0
MOVL C00742 V=800.0 PL=0
MOVL C00743 V=800.0 PL=0
MOVL C00744 V=800.0 PL=0
MOVL C00745 V=800.0 PL=0
MOVL C00746 V=800.0 PL=0
MOVL C00747 V=800.0 PL=0
MOVL C00748 V=800.0 PL=0
MOVL C00749 V=800.0 PL=0
MOVL C00750 V=800.0 PL=0
MOVL C00751 V=800.0 PL=0
MOVL C00752 V=800.0 PL=0
MOVL C00753 V=800.0 PL=0
MOVL C00754 V=800.0 PL=0
MOVL C00755 V=800.0 PL=0
MOVL C00756 V=800.0 PL=0
MOVL C00757 V=800.0 PL=0
MOVL C00758 V=800.0 PL=0
MOVL C00759 V=800.0 PL=0
MOVL C00760 V=800.0 PL=0
MOVL C00761 V=800.0 PL=0
MOVL C00762 V=800.0 PL=0
MOVL C00763 V=800.0 PL=0
MOVL C00764 V=800.0 PL=0
MOVL C00765 V=800.0 PL=0
MOVL C00766 V=800.0 PL=0
MOVL C00767 V=800.0 PL=0
MOVL C00768 V=800.0 PL=0
MOVL C00769 V=800.0 PL=0
MOVL C00770 V=800.0 PL=0
MOVL C00771 V=800.0 PL=0
MOVL C00772 V=800.0 PL=0
MOVL C00773 V=800.0 PL=0
MOVL C00774 V=800.0 PL=0
MOVL C00775 V=800.0 PL=0
MOVL C00776 V=800.0 PL=0
MOVL C00777 V=800.0 PL=0
MOVL C00778 V=800.0 PL=0
MOVL C00779 V=800.0 PL=0
MOVL C00780 V=800.0 PL=0
MOVL C00781 V=800.0 PL=0
MOVL C00782 V=800.0 PL=0
MOVL C00783 V=800.0 PL=0
MOVL C00784 V=800.0 PL=0
MOVL C00785 V=800.0 PL=0
MOVL C00786 V=800.0 PL=0
MOVL C00787 V=800.0 PL=0
MOVL C00788 V=800.0 PL=0
MOVL C00789 V=800.0 PL=0
MOVL C00790 V=800.0 PL=0
MOVL C00791 V=800.0 PL=0
MOVL C00792 V=800.0 PL=0
MOVL C00793 V=800.0 PL=0
MOVL C00794 V=800.0 PL=0
MOVL C00795 V=800.0 PL=0
MOVL C00796 V=800.0 PL=0
MOVL C00797 V=800.0 PL=0
MOVL C00798 V=800.0 PL=0
MOVL C00799 V=800.0 PL=0
MOVL C00800 V=800.0 PL=0
MOVL C00801 V=800.0 PL=0
MOVL C00802 V=800.0 PL=0
MOVL C00803 V=800.0 PL=0
MOVL C00804 V=800.0 PL=0
MOVL C00805 V=800.0 PL=0
MOVL C00806 V=800.0 PL=0
MOVL C00807 V=800.0 PL=0
MOVL C00808 V=800.0 PL=0
MOVL C00809 V=800.0 PL=0
MOVL C00810 V=800.0 PL=0
MOVL C00811 V=800.0 PL=0
MOVL C00812 V=800.0 PL=0
MOVL C00813 V=800.0 PL=0
MOVL C00814 V=800.0 PL=0
MOVL C00815 V=800.0 PL=0
MOVL C00816 V=800.0 PL=0
MOVL C00817 V=800.0 PL=0
MOVL C00818 V=800.0 PL=0
MOVL C00819 V=800.0 PL=0
MOVL C00820 V=800.0 PL=0
MOVL C00821 V=800.0 PL=0
MOVL C00822 V=800.0 PL=0
MOVL C00823 V=800.0 PL=0
MOVL C00824 V=800.0 PL=0
MOVL C00825 V=800.0 PL=0
MOVL C00826 V=800.0 PL=0
MOVL C00827 V=800.0 PL=0
MOVL C00828 V=800.0 PL=0
MOVL C00829 V=800.0 PL=0
MOVL C00830 V=800.0 PL=0
MOVL C00831 V=800.0 PL=0
MOVL C00832 V=800.0 PL=0
MOVL C00833 V=800.0 PL=0
MOVL C00834 V=800.0 PL=0
MOVL C00835 V=800.0 PL=0
MOVL C00836 V=800.0 PL=0
MOVL C00837 V=800.0 PL=0
MOVL C00838 V=800.0 PL=0
MOVL C00839 V=800.0 PL=0
MOVL C00840 V=800.0 PL=0
MOVL C00841 V=800.0 PL=0
MOVL C00842 V=800.0 PL=0
MOVL C00843 V=800.0 PL=0
MOVL C00844 V=800.0 PL=0
MOVL C00845 V=800.0 PL=0
MOVL C00846 V=800.0 PL=0
MOVL C00847 V=800.0 PL=0
MOVL C00848 V=800.0 PL=0
MOVL C00849 V=800.0 PL=0
MOVL C00850 V=800.0 PL=0
MOVL C00851 V=800.0 PL=0
MOVL C00852 V=800.0 PL=0
MOVL C00853 V=800.0 PL=0
MOVL C00854 V=800.0 PL=0
MOVL C00855 V=800.0 PL=0
MOVL C00856 V=800.0 PL=0
MOVL C00857 V=800.0 PL=0
MOVL C00858 V=800.0 PL=0
MOVL C00859 V=800.0 PL=0
MOVL C00860 V=800.0 PL=0
MOVL C00861 V=800.0 PL=0
MOVL C00862 V=800.0 PL=0
MOVL C00863 V=800.0 PL=0
MOVL C00864 V=800.0 PL=0
MOVL C00865 V=800.0 PL=0
MOVL C00866 V=800.0 PL=0
MOVL C00867 V=800.0 PL=0
MOVL C00868 V=800.0 PL=0
MOVL C00869 V=800.0 PL=0
MOVL C00870 V=800.0 PL=0
MOVL C00871 V=800.0 PL=0
MOVL C00872 V=800.0 PL=0
MOVL C00873 V=800.0 PL=0
MOVL C00874 V=800.0 PL=0
MOVL C00875 V=800.0 PL=0
MOVL C00876 V=800.0 PL=0
MOVL C00877 V=800.0 PL=0
MOVL C00878 V=800.0 PL=0
MOVL C00879 V=800.0 PL=0
MOVL C00880 V=800.0 PL=0
MOVL C00881 V=800.0 PL=0
MOVL C00882 V=800.0 PL=0
MOVL C00883 V=800.0 PL=0
MOVL C00884 V=800.0 PL=0
MOVL C00885 V=800.0 PL=0
MOVL C00886 V=800.0 PL=0
MOVL C00887 V=800.0 PL=0
MOVL C00888 V=800.0 PL=0
MOVL C00889 V=800.0 PL=0
MOVL C00890 V=800.0 PL=0
MOVL C00891 V=800.0 PL=0
MOVL C00892 V=800.0 PL=0
MOVL C00893 V=800.0 PL=0
MOVL C00894 V=800.0 PL=0
MOVL C00895 V=800.0 PL=0
MOVL C00896 V=800.0 PL=0
MOVL C00897 V=800.0 PL=0
MOVL C00898 V=800.0 PL=0
MOVL C00899 V=800.0 PL=0
MOVL C00900 V=800.0 PL=0
MOVL C00901 V=800.0 PL=0
MOVL C00902 V=800.0 PL=0
MOVL C00903 V=800.0 PL=0
MOVL C00904 V=800.0 PL=0
MOVL C00905 V=800.0 PL=0
MOVL C00906 V=800.0 PL=0
MOVL C00907 V=800.0 PL=0
MOVL C00908 V=800.0 PL=0
MOVL C00909 V=800.0 PL=0
MOVL C00910 V=800.0 PL=0
MOVL C00911 V=800.0 PL=0
MOVL C00912 V=800.0 PL=0
MOVL C00913 V=800.0 PL=0
MOVL C00914 V=800.0 PL=0
MOVL C00915 V=800.0 PL=0
MOVL C00916 V=800.0 PL=0
MOVL C00917 V=800.0 PL=0
MOVL C00918 V=800.0 PL=0
MOVL C00919 V=800.0 PL=0
MOVL C00920 V=800.0 PL=0
MOVL C00921 V=800.0 PL=0
MOVL C00922 V=800.0 PL=0
MOVL C00923 V=800.0 PL=0
MOVL C00924 V=800.0 PL=0
MOVL C00925 V=800.0 PL=0
MOVL C00926 V=800.0 PL=0
MOVL C00927 V=800.0 PL=0
MOVL C00928 V=800.0 PL=0
MOVL C00929 V=800.0 PL=0
MOVL C00930 V=800.0 PL=0
MOVL C00931 V=800.0 PL=0
MOVL C00932 V=800.0 PL=0
MOVL C00933 V=800.0 PL=0
MOVL C00934 V=800.0 PL=0
MOVL C00935 V=800.0 PL=0
MOVL C00936 V=800.0 PL=0
MOVL C00937 V=800.0 PL=0
MOVL C00938 V=800.0 PL=0
MOVL C00939 V=800.0 PL=0
MOVL C00940 V=800.0 PL=0
MOVL C00941 V=800.0 PL=0
MOVL C00942 V=800.0 PL=0
MOVL C00943 V=800.0 PL=0
MOVL C00944 V=800.0 PL=0
MOVL C00945 V=800.0 PL=0
MOVL C00946 V=800.0 PL=0
MOVL C00947 V=800.0 PL=0
MOVL C00948 V=800.0 PL=0
MOVL C00949 V=800.0 PL=0
MOVL C00950 V=800.0 PL=0
MOVL C00951 V=800.0 PL=0
MOVL C00952 V=800.0 PL=0
MOVL C00953 V=800.0 PL=0
MOVL C00954 V=800.0 PL=0
MOVL C00955 V=800.0 PL=0
MOVL C00956 V=800.0 PL=0
MOVL C00957 V=800.0 PL=0
MOVL C00958 V=800.0 PL=0
MOVL C00959 V=800.0 PL=0
MOVL C00960 V=800.0 PL=0
MOVL C00961 V=800.0 PL=0
MOVL C00962 V=800.0 PL=0
MOVL C00963 V=800.0 PL=0
MOVL C00964 V=800.0 PL=0
MOVL C00965 V=800.0 PL=0
MOVL C00966 V=800.0 PL=0
MOVL C00967 V=800.0 PL=0
MOVL C00968 V=800.0 PL=0
MOVL C00969 V=800.0 PL=0
MOVL C00970 V=800.0 PL=0
MOVL C00971 V=800.0 PL=0
MOVL C00972 V=800.0 PL=0
MOVL C00973 V=800.0 PL=0
MOVL C00974 V=800.0 PL=0
MOVL C00975 V=800.0 PL=0
MOVL C00976 V=800.0 PL=0
MOVL C00977 V=800.0 PL=0
MOVL C00978 V=800.0 PL=0
MOVL C00979 V=800.0 PL=0
MOVL C00980 V=800.0 PL=0
MOVL C00981 V=800.0 PL=0
MOVL C00982 V=800.0 PL=0
MOVL C00983 V=800.0 PL=0
MOVL C00984 V=800.0 PL=0
MOVL C00985 V=800.0 PL=0
MOVL C00986 V=800.0 PL=0
MOVL C00987 V=800.0 PL=0
MOVL C00988 V=800.0 PL=0
MOVL C00989 V=800.0 PL=0
MOVL C00990 V=800.0 PL=0
MOVL C00991 V=800.0 PL=0
MOVL C00992 V=800.0 PL=0
MOVL C00993 V=800.0 PL=0
MOVL C00994 V=800.0 PL=0
MOVL C00995 V=800.0 PL=0
MOVL C00996 V=800.0 PL=0
MOVL C00997 V=800.0 PL=0
MOVL C00998 V=800.0 PL=0
MOVL C00999 V=800.0 PL=0
MOVL C01000 V=800.0 PL=0
MOVL C01001 V=800.0 PL=0
MOVL C01002 V=800.0 PL=0
MOVL C01003 V=800.0 PL=0
MOVL C01004 V=800.0 PL=0
MOVL C01005 V=800.0 PL=0
MOVL C01006 V=800.0 PL=0
MOVL C01007 V=800.0 PL=0
MOVL C01008 V=800.0 PL=0
MOVL C01009 V=800.0 PL=0
MOVL C01010 V=800.0 PL=0
MOVL C01011 V=800.0 PL=0
MOVL C01012 V=800.0 PL=0
MOVL C01013 V=800.0 PL=0
MOVL C01014 V=800.0 PL=0
MOVL C01015 V=800.0 PL=0
MOVL C01016 V=800.0 PL=0
MOVL C01017 V=800.0 PL=0
MOVL C01018 V=800.0 PL=0
MOVL C01019 V=800.0 PL=0
MOVL C01020 V=800.0 PL=0
MOVL C01021 V=800.0 PL=0
MOVL C01022 V=800.0 PL=0
MOVL C01023 V=800.0 PL=0
MOVL C01024 V=800.0 PL=0
MOVL C01025 V=800.0 PL=0
MOVL C01026 V=800.0 PL=0
MOVL C01027 V=800.0 PL=0
MOVL C01028 V=800.0 PL=0
MOVL C01029 V=800.0 PL=0
MOVL C01030 V=800.0 PL=0
MOVL C01031 V=800.0 PL=0
MOVL C01032 V=800.0 PL=0
MOVL C01033 V=800.0 PL=0
MOVL C01034 V=800.0 PL=0
MOVL C01035 V=800.0 PL=0
MOVL C01036 V=800.0 PL=0
MOVL C01037 V=800.0 PL=0
MOVL C01038 V=800.0 PL=0
MOVL C01039 V=800.0 PL=0
MOVL C01040 V=800.0 PL=0
MOVL C01041 V=800.0 PL=0
MOVL C01042 V=800.0 PL=0
MOVL C01043 V=800.0 PL=0
MOVL C01044 V=800.0 PL=0
MOVL C01045 V=800.0 PL=0
MOVL C01046 V=800.0 PL=0
MOVL C01047 V=800.0 PL=0
MOVL C01048 V=800.0 PL=0
MOVL C01049 V=800.0 PL=0
MOVL C01050 V=800.0 PL=0
MOVL C01051 V=800.0 PL=0
MOVL C01052 V=800.0 PL=0
MOVL C01053 V=800.0 PL=0
MOVL C01054 V=800.0 PL=0
MOVL C01055 V=800.0 PL=0
MOVL C01056 V=800.0 PL=0
MOVL C01057 V=800.0 PL=0
MOVL C01058 V=800.0 PL=0
MOVL C01059 V=800.0 PL=0
MOVL C01060 V=800.0 PL=0
MOVL C01061 V=800.0 PL=0
MOVL C01062 V=800.0 PL=0
MOVL C01063 V=800.0 PL=0
MOVL C01064 V=800.0 PL=0
MOVL C01065 V=800.0 PL=0
MOVL C01066 V=800.0 PL=0
MOVL C01067 V=800.0 PL=0
MOVL C01068 V=800.0 PL=0
MOVL C01069 V=800.0 PL=0
MOVL C01070 V=800.0 PL=0
MOVL C01071 V=800.0 PL=0
MOVL C01072 V=800.0 PL=0
MOVL C01073 V=800.0 PL=0
MOVL C01074 V=800.0 PL=0
MOVL C01075 V=800.0 PL=0
MOVL C01076 V=800.0 PL=0
MOVL C01077 V=800.0 PL=0
MOVL C01078 V=800.0 PL=0
MOVL C01079 V=800.0 PL=0
MOVL C01080 V=800.0 PL=0
MOVL C01081 V=800.0 PL=0
MOVL C01082 V=800.0 PL=0
MOVL C01083 V=800.0 PL=0
MOVL C01084 V=800.0 PL=0
MOVL C01085 V=800.0 PL=0
MOVL C01086 V=800.0 PL=0
MOVL C01087 V=800.0 PL=0
MOVL C01088 V=800.0 PL=0
MOVL C01089 V=800.0 PL=0
MOVL C01090 V=800.0 PL=0
MOVL C01091 V=800.0 PL=0
MOVL C01092 V=800.0 PL=0
MOVL C01093 V=800.0 PL=0
MOVL C01094 V=800.0 PL=0
MOVL C01095 V=800.0 PL=0
MOVL C01096 V=800.0 PL=0
MOVL C01097 V=800.0 PL=0
MOVL C01098 V=800.0 PL=0
MOVL C01099 V=800.0 PL=0
MOVL C01100 V=800.0 PL=0
MOVL C01101 V=800.0 PL=0
MOVL C01102 V=800.0 PL=0
MOVL C01103 V=800.0 PL=0
MOVL C01104 V=800.0 PL=0
MOVL C01105 V=800.0 PL=0
MOVL C01106 V=800.0 PL=0
MOVL C01107 V=800.0 PL=0
MOVL C01108 V=800.0 PL=0
MOVL C01109 V=800.0 PL=0
MOVL C01110 V=800.0 PL=0
MOVL C01111 V=800.0 PL=0
MOVL C01112 V=800.0 PL=0
MOVL C01113 V=800.0 PL=0
MOVL C01114 V=800.0 PL=0
MOVL C01115 V=800.0 PL=0
MOVL C01116 V=800.0 PL=0
MOVL C01117 V=800.0 PL=0
MOVL C01118 V=800.0 PL=0
MOVL C01119 V=800.0 PL=0
MOVL C01120 V=800.0 PL=0
MOVL C01121 V=800.0 PL=0
MOVL C01122 V=800.0 PL=0
MOVL C01123 V=800.0 PL=0
MOVL C01124 V=800.0 PL=0
MOVL C01125 V=800.0 PL=0
MOVL C01126 V=800.0 PL=0
MOVL C01127 V=800.0 PL=0
MOVL C01128 V=800.0 PL=0
MOVL C01129 V=800.0 PL=0
MOVL C01130 V=800.0 PL=0
MOVL C01131 V=800.0 PL=0
MOVL C01132 V=800.0 PL=0
MOVL C01133 V=800.0 PL=0
MOVL C01134 V=800.0 PL=0
MOVL C01135 V=800.0 PL=0
MOVL C01136 V=800.0 PL=0
MOVL C01137 V=800.0 PL=0
MOVL C01138 V=800.0 PL=0
MOVL C01139 V=800.0 PL=0
MOVL C01140 V=800.0 PL=0
MOVL C01141 V=800.0 PL=0
MOVL C01142 V=800.0 PL=0
MOVL C01143 V=800.0 PL=0
MOVL C01144 V=800.0 PL=0
MOVL C01145 V=800.0 PL=0
MOVL C01146 V=800.0 PL=0
MOVL C01147 V=800.0 PL=0
MOVL C01148 V=800.0 PL=0
MOVL C01149 V=800.0 PL=0
MOVL C01150 V=800.0 PL=0
MOVL C01151 V=800.0 PL=0
MOVL C01152 V=800.0 PL=0
MOVL C01153 V=800.0 PL=0
MOVL C01154 V=800.0 PL=0
MOVL C01155 V=800.0 PL=0
MOVL C01156 V=800.0 PL=0
MOVL C01157 V=800.0 PL=0
MOVL C01158 V=800.0 PL=0
MOVL C01159 V=800.0 PL=0
MOVL C01160 V=800.0 PL=0
MOVL C01161 V=800.0 PL=0
MOVL C01162 V=800.0 PL=0
MOVL C01163 V=800.0 PL=0
MOVL C01164 V=800.0 PL=0
MOVL C01165 V=800.0 PL=0
MOVL C01166 V=800.0 PL=0
MOVL C01167 V=800.0 PL=0
MOVL C01168 V=800.0 PL=0
MOVL C01169 V=800.0 PL=0
MOVL C01170 V=800.0 PL=0
MOVL C01171 V=800.0 PL=0
MOVL C01172 V=800.0 PL=0
MOVL C01173 V=800.0 PL=0
MOVL C01174 V=800.0 PL=0
MOVL C01175 V=800.0 PL=0
MOVL C01176 V=800.0 PL=0
MOVL C01177 V=800.0 PL=0
MOVL C01178 V=800.0 PL=0
MOVL C01179 V=800.0 PL=0
MOVL C01180 V=800.0 PL=0
MOVL C01181 V=800.0 PL=0
MOVL C01182 V=800.0 PL=0
MOVL C01183 V=800.0 PL=0
MOVL C01184 V=800.0 PL=0
MOVL C01185 V=800.0 PL=0
MOVL C01186 V=800.0 PL=0
MOVL C01187 V=800.0 PL=0
MOVL C01188 V=800.0 PL=0
MOVL C01189 V=800.0 PL=0
MOVL C01190 V=800.0 PL=0
MOVL C01191 V=800.0 PL=0
MOVL C01192 V=800.0 PL=0
MOVL C01193 V=800.0 PL=0
MOVL C01194 V=800.0 PL=0
MOVL C01195 V=800.0 PL=0
MOVL C01196 V=800.0 PL=0
MOVL C01197 V=800.0 PL=0
MOVL C01198 V=800.0 PL=0
MOVL C01199 V=800.0 PL=0
MOVL C01200 V=800.0 PL=0
MOVL C01201 V=800.0 PL=0
MOVL C01202 V=800.0 PL=0
MOVL C01203 V=800.0 PL=0
MOVL C01204 V=800.0 PL=0
MOVL C01205 V=800.0 PL=0
MOVL C01206 V=800.0 PL=0
MOVL C01207 V=800.0 PL=0
MOVL C01208 V=800.0 PL=0
MOVL C01209 V=800.0 PL=0
MOVL C01210 V=800.0 PL=0
MOVL C01211 V=800.0 PL=0
MOVL C01212 V=800.0 PL=0
MOVL C01213 V=800.0 PL=0
MOVL C01214 V=800.0 PL=0
MOVL C01215 V=800.0 PL=0
MOVL C01216 V=800.0 PL=0
MOVL C01217 V=800.0 PL=0
MOVL C01218 V=800.0 PL=0
MOVL C01219 V=800.0 PL=0
MOVL C01220 V=800.0 PL=0
MOVL C01221 V=800.0 PL=0
MOVL C01222 V=800.0 PL=0
MOVL C01223 V=800.0 PL=0
MOVL C01224 V=800.0 PL=0
MOVL C01225 V=800.0 PL=0
MOVL C01226 V=800.0 PL=0
MOVL C01227 V=800.0 PL=0
MOVL C01228 V=800.0 PL=0
MOVL C01229 V=800.0 PL=0
MOVL C01230 V=800.0 PL=0
MOVL C01231 V=800.0 PL=0
MOVL C01232 V=800.0 PL=0
MOVL C01233 V=800.0 PL=0
MOVL C01234 V=800.0 PL=0
MOVL C01235 V=800.0 PL=0
MOVL C01236 V=800.0 PL=0
MOVL C01237 V=800.0 PL=0
MOVL C01238 V=800.0 PL=0
MOVL C01239 V=800.0 PL=0
MOVL C01240 V=800.0 PL=0
MOVL C01241 V=800.0 PL=0
MOVL C01242 V=800.0 PL=0
MOVL C01243 V=800.0 PL=0
MOVL C01244 V=800.0 PL=0
MOVL C01245 V=800.0 PL=0
MOVL C01246 V=800.0 PL=0
MOVL C01247 V=800.0 PL=0
MOVL C01248 V=800.0 PL=0
MOVL C01249 V=800.0 PL=0
MOVL C01250 V=800.0 PL=0
MOVL C01251 V=800.0 PL=0
MOVL C01252 V=800.0 PL=0
MOVL C01253 V=800.0 PL=0
MOVL C01254 V=800.0 PL=0
MOVL C01255 V=800.0 PL=0
MOVL C01256 V=800.0 PL=0
MOVL C01257 V=800.0 PL=0
MOVL C01258 V=800.0 PL=0
MOVL C01259 V=800.0 PL=0
MOVL C01260 V=800.0 PL=0
MOVL C01261 V=800.0 PL=0
MOVL C01262 V=800.0 PL=0
MOVL C01263 V=800.0 PL=0
MOVL C01264 V=800.0 PL=0
MOVL C01265 V=800.0 PL=0
MOVL C01266 V=800.0 PL=0
MOVL C01267 V=800.0 PL=0
MOVL C01268 V=800.0 PL=0
MOVL C01269 V=800.0 PL=0
MOVL C01270 V=800.0 PL=0
MOVL C01271 V=800.0 PL=0
MOVL C01272 V=800.0 PL=0
MOVL C01273 V=800.0 PL=0
MOVL C01274 V=800.0 PL=0
MOVL C01275 V=800.0 PL=0
MOVL C01276 V=800.0 PL=0
MOVL C01277 V=800.0 PL=0
MOVL C01278 V=800.0 PL=0
MOVL C01279 V=800.0 PL=0
MOVL C01280 V=800.0 PL=0
MOVL C01281 V=800.0 PL=0
MOVL C01282 V=800.0 PL=0
MOVL C01283 V=800.0 PL=0
MOVL C01284 V=800.0 PL=0
MOVL C01285 V=800.0 PL=0
MOVL C01286 V=800.0 PL=0
MOVL C01287 V=800.0 PL=0
MOVL C01288 V=800.0 PL=0
MOVL C01289 V=800.0 PL=0
MOVL C01290 V=800.0 PL=0
MOVL C01291 V=800.0 PL=0
MOVL C01292 V=800.0 PL=0
MOVL C01293 V=800.0 PL=0
MOVL C01294 V=800.0 PL=0
MOVL C01295 V=800.0 PL=0
MOVL C01296 V=800.0 PL=0
MOVL C01297 V=800.0 PL=0
MOVL C01298 V=800.0 PL=0
MOVL C01299 V=800.0 PL=0
MOVL C01300 V=800.0 PL=0
MOVL C01301 V=800.0 PL=0
MOVL C01302 V=800.0 PL=0
MOVL C01303 V=800.0 PL=0
MOVL C01304 V=800.0 PL=0
MOVL C01305 V=800.0 PL=0
MOVL C01306 V=800.0 PL=0
MOVL C01307 V=800.0 PL=0
MOVL C01308 V=800.0 PL=0
MOVL C01309 V=800.0 PL=0
MOVL C01310 V=800.0 PL=0
MOVL C01311 V=800.0 PL=0
MOVL C01312 V=800.0 PL=0
MOVL C01313 V=800.0 PL=0
MOVL C01314 V=800.0 PL=0
MOVL C01315 V=800.0 PL=0
MOVL C01316 V=800.0 PL=0
MOVL C01317 V=800.0 PL=0
MOVL C01318 V=800.0 PL=0
MOVL C01319 V=800.0 PL=0
MOVL C01320 V=800.0 PL=0
MOVL C01321 V=800.0 PL=0
MOVL C01322 V=800.0 PL=0
MOVL C01323 V=800.0 PL=0
MOVL C01324 V=800.0 PL=0
MOVL C01325 V=800.0 PL=0
MOVL C01326 V=800.0 PL=0
MOVL C01327 V=800.0 PL=0
MOVL C01328 V=800.0 PL=0
MOVL C01329 V=800.0 PL=0
MOVL C01330 V=800.0 PL=0
MOVL C01331 V=800.0 PL=0
MOVL C01332 V=800.0 PL=0
MOVL C01333 V=800.0 PL=0
MOVL C01334 V=800.0 PL=0
MOVL C01335 V=800.0 PL=0
MOVL C01336 V=800.0 PL=0
MOVL C01337 V=800.0 PL=0
MOVL C01338 V=800.0 PL=0
MOVL C01339 V=800.0 PL=0
MOVL C01340 V=800.0 PL=0
MOVL C01341 V=800.0 PL=0
MOVL C01342 V=800.0 PL=0
MOVL C01343 V=800.0 PL=0
MOVL C01344 V=800.0 PL=0
MOVL C01345 V=800.0 PL=0
MOVL C01346 V=800.0 PL=0
MOVL C01347 V=800.0 PL=0
MOVL C01348 V=800.0 PL=0
MOVL C01349 V=800.0 PL=0
MOVL C01350 V=800.0 PL=0
MOVL C01351 V=800.0 PL=0
MOVL C01352 V=800.0 PL=0
MOVL C01353 V=800.0 PL=0
MOVL C01354 V=800.0 PL=0
MOVL C01355 V=800.0 PL=0
MOVL C01356 V=800.0 PL=0
MOVL C01357 V=800.0 PL=0
MOVL C01358 V=800.0 PL=0
MOVL C01359 V=800.0 PL=0
MOVL C01360 V=800.0 PL=0
MOVL C01361 V=800.0 PL=0
MOVL C01362 V=800.0 PL=0
MOVL C01363 V=800.0 PL=0
MOVL C01364 V=800.0 PL=0
MOVL C01365 V=800.0 PL=0
MOVL C01366 V=800.0 PL=0
MOVL C01367 V=800.0 PL=0
MOVL C01368 V=800.0 PL=0
MOVL C01369 V=800.0 PL=0
MOVL C01370 V=800.0 PL=0
MOVL C01371 V=800.0 PL=0
MOVL C01372 V=800.0 PL=0
MOVL C01373 V=800.0 PL=0
MOVL C01374 V=800.0 PL=0
MOVL C01375 V=800.0 PL=0
MOVL C01376 V=800.0 PL=0
MOVL C01377 V=800.0 PL=0
MOVL C01378 V=800.0 PL=0
MOVL C01379 V=800.0 PL=0
MOVL C01380 V=800.0 PL=0
MOVL C01381 V=800.0 PL=0
MOVL C01382 V=800.0 PL=0
MOVL C01383 V=800.0 PL=0
MOVL C01384 V=800.0 PL=0
MOVL C01385 V=800.0 PL=0
MOVL C01386 V=800.0 PL=0
MOVL C01387 V=800.0 PL=0
MOVL C01388 V=800.0 PL=0
MOVL C01389 V=800.0 PL=0
MOVL C01390 V=800.0 PL=0
MOVL C01391 V=800.0 PL=0
MOVL C01392 V=800.0 PL=0
MOVL C01393 V=800.0 PL=0
MOVL C01394 V=800.0 PL=0
MOVL C01395 V=800.0 PL=0
MOVL C01396 V=800.0 PL=0
MOVL C01397 V=800.0 PL=0
MOVL C01398 V=800.0 PL=0
MOVL C01399 V=800.0 PL=0
MOVL C01400 V=800.0 PL=0
MOVL C01401 V=800.0 PL=0
MOVL C01402 V=800.0 PL=0
MOVL C01403 V=800.0 PL=0
MOVL C01404 V=800.0 PL=0
MOVL C01405 V=800.0 PL=0
MOVL C01406 V=800.0 PL=0
MOVL C01407 V=800.0 PL=0
MOVL C01408 V=800.0 PL=0
MOVL C01409 V=800.0 PL=0
MOVL C01410 V=800.0 PL=0
MOVL C01411 V=800.0 PL=0
MOVL C01412 V=800.0 PL=0
MOVL C01413 V=800.0 PL=0
MOVL C01414 V=800.0 PL=0
MOVL C01415 V=800.0 PL=0
MOVL C01416 V=800.0 PL=0
MOVL C01417 V=800.0 PL=0
MOVL C01418 V=800.0 PL=0
MOVL C01419 V=800.0 PL=0
MOVL C01420 V=800.0 PL=0
MOVL C01421 V=800.0 PL=0
MOVL C01422 V=800.0 PL=0
MOVL C01423 V=800.0 PL=0
MOVL C01424 V=800.0 PL=0
MOVL C01425 V=800.0 PL=0
MOVL C01426 V=800.0 PL=0
MOVL C01427 V=800.0 PL=0
MOVL C01428 V=800.0 PL=0
MOVL C01429 V=800.0 PL=0
MOVL C01430 V=800.0 PL=0
MOVL C01431 V=800.0 PL=0
MOVL C01432 V=800.0 PL=0
MOVL C01433 V=800.0 PL=0
MOVL C01434 V=800.0 PL=0
MOVL C01435 V=800.0 PL=0
MOVL C01436 V=800.0 PL=0
MOVL C01437 V=800.0 PL=0
MOVL C01438 V=800.0 PL=0
MOVL C01439 V=800.0 PL=0
MOVL C01440 V=800.0 PL=0
MOVL C01441 V=800.0 PL=0
MOVL C01442 V=800.0 PL=0
MOVL C01443 V=800.0 PL=0
MOVL C01444 V=800.0 PL=0
MOVL C01445 V=800.0 PL=0
MOVL C01446 V=800.0 PL=0
MOVL C01447 V=800.0 PL=0
MOVL C01448 V=800.0 PL=0
MOVL C01449 V=800.0 PL=0
MOVL C01450 V=800.0 PL=0
MOVL C01451 V=800.0 PL=0
MOVL C01452 V=800.0 PL=0
MOVL C01453 V=800.0 PL=0
MOVL C01454 V=800.0 PL=0
MOVL C01455 V=800.0 PL=0
MOVL C01456 V=800.0 PL=0
MOVL C01457 V=800.0 PL=0
MOVL C01458 V=800.0 PL=0
MOVL C01459 V=800.0 PL=0
MOVL C01460 V=800.0 PL=0
MOVL C01461 V=800.0 PL=0
MOVL C01462 V=800.0 PL=0
MOVL C01463 V=800.0 PL=0
MOVL C01464 V=800.0 PL=0
MOVL C01465 V=800.0 PL=0
MOVL C01466 V=800.0 PL=0
MOVL C01467 V=800.0 PL=0
MOVL C01468 V=800.0 PL=0
MOVL C01469 V=800.0 PL=0
MOVL C01470 V=800.0 PL=0
MOVL C01471 V=800.0 PL=0
MOVL C01472 V=800.0 PL=0
MOVL C01473 V=800.0 PL=0
MOVL C01474 V=800.0 PL=0
MOVL C01475 V=800.0 PL=0
MOVL C01476 V=800.0 PL=0
MOVL C01477 V=800.0 PL=0
MOVL C01478 V=800.0 PL=0
MOVL C01479 V=800.0 PL=0
MOVL C01480 V=800.0 PL=0
MOVL C01481 V=800.0 PL=0
MOVL C01482 V=800.0 PL=0
MOVL C01483 V=800.0 PL=0
MOVL C01484 V=800.0 PL=0
MOVL C01485 V=800.0 PL=0
MOVL C01486 V=800.0 PL=0
MOVL C01487 V=800.0 PL=0
MOVL C01488 V=800.0 PL=0
MOVL C01489 V=800.0 PL=0
MOVL C01490 V=800.0 PL=0
MOVL C01491 V=800.0 PL=0
MOVL C01492 V=800.0 PL=0
MOVL C01493 V=800.0 PL=0
MOVL C01494 V=800.0 PL=0
MOVL C01495 V=800.0 PL=0
MOVL C01496 V=800.0 PL=0
MOVL C01497 V=800.0 PL=0
MOVL C01498 V=800.0 PL=0
MOVL C01499 V=800.0 PL=0
MOVL C01500 V=800.0 PL=0
MOVL C01501 V=800.0 PL=0
MOVL C01502 V=800.0 PL=0
MOVL C01503 V=800.0 PL=0
MOVL C01504 V=800.0 PL=0
MOVL C01505 V=800.0 PL=0
MOVL C01506 V=800.0 PL=0
MOVL C01507 V=800.0 PL=0
MOVL C01508 V=800.0 PL=0
MOVL C01509 V=800.0 PL=0
MOVL C01510 V=800.0 PL=0
MOVL C01511 V=800.0 PL=0
MOVL C01512 V=800.0 PL=0
MOVL C01513 V=800.0 PL=0
MOVL C01514 V=800.0 PL=0
MOVL C01515 V=800.0 PL=0
MOVL C01516 V=800.0 PL=0
MOVL C01517 V=800.0 PL=0
MOVL C01518 V=800.0 PL=0
MOVL C01519 V=800.0 PL=0
MOVL C01520 V=800.0 PL=0
MOVL C01521 V=800.0 PL=0
MOVL C01522 V=800.0 PL=0
MOVL C01523 V=800.0 PL=0
MOVL C01524 V=800.0 PL=0
MOVL C01525 V=800.0 PL=0
MOVL C01526 V=800.0 PL=0
MOVL C01527 V=800.0 PL=0
MOVL C01528 V=800.0 PL=0
MOVL C01529 V=800.0 PL=0
MOVL C01530 V=800.0 PL=0
MOVL C01531 V=800.0 PL=0
MOVL C01532 V=800.0 PL=0
MOVL C01533 V=800.0 PL=0
MOVL C01534 V=800.0 PL=0
MOVL C01535 V=800.0 PL=0
MOVL C01536 V=800.0 PL=0
MOVL C01537 V=800.0 PL=0
MOVL C01538 V=800.0 PL=0
MOVL C01539 V=800.0 PL=0
MOVL C01540 V=800.0 PL=0
MOVL C01541 V=800.0 PL=0
MOVL C01542 V=800.0 PL=0
MOVL C01543 V=800.0 PL=0
MOVL C01544 V=800.0 PL=0
MOVL C01545 V=800.0 PL=0
MOVL C01546 V=800.0 PL=0
MOVL C01547 V=800.0 PL=0
MOVL C01548 V=800.0 PL=0
MOVL C01549 V=800.0 PL=0
MOVL C01550 V=800.0 PL=0
MOVL C01551 V=800.0 PL=0
MOVL C01552 V=800.0 PL=0
MOVL C01553 V=800.0 PL=0
MOVL C01554 V=800.0 PL=0
MOVL C01555 V=800.0 PL=0
MOVL C01556 V=800.0 PL=0
MOVL C01557 V=800.0 PL=0
MOVL C01558 V=800.0 PL=0
MOVL C01559 V=800.0 PL=0
MOVL C01560 V=800.0 PL=0
MOVL C01561 V=800.0 PL=0
MOVL C01562 V=800.0 PL=0
MOVL C01563 V=800.0 PL=0
MOVL C01564 V=800.0 PL=0
MOVL C01565 V=800.0 PL=0
MOVL C01566 V=800.0 PL=0
MOVL C01567 V=800.0 PL=0
MOVL C01568 V=800.0 PL=0
MOVL C01569 V=800.0 PL=0
MOVL C01570 V=800.0 PL=0
MOVL C01571 V=800.0 PL=0
MOVL C01572 V=800.0 PL=0
MOVL C01573 V=800.0 PL=0
MOVL C01574 V=800.0 PL=0
MOVL C01575 V=800.0 PL=0
MOVL C01576 V=800.0 PL=0
MOVL C01577 V=800.0 PL=0
MOVL C01578 V=800.0 PL=0
MOVL C01579 V=800.0 PL=0
MOVL C01580 V=800.0 PL=0
MOVL C01581 V=800.0 PL=0
MOVL C01582 V=800.0 PL=0
MOVL C01583 V=800.0 PL=0
MOVL C01584 V=800.0 PL=0
MOVL C01585 V=800.0 PL=0
MOVL C01586 V=800.0 PL=0
MOVL C01587 V=800.0 PL=0
MOVL C01588 V=800.0 PL=0
MOVL C01589 V=800.0 PL=0
MOVL C01590 V=800.0 PL=0
MOVL C01591 V=800.0 PL=0
MOVL C01592 V=800.0 PL=0
MOVL C01593 V=800.0 PL=0
MOVL C01594 V=800.0 PL=0
MOVL C01595 V=800.0 PL=0
MOVL C01596 V=800.0 PL=0
MOVL C01597 V=800.0 PL=0
MOVL C01598 V=800.0 PL=0
MOVL C01599 V=800.0 PL=0
MOVL C01600 V=800.0 PL=0
MOVL C01601 V=800.0 PL=0
MOVL C01602 V=800.0 PL=0
MOVL C01603 V=800.0 PL=0
MOVL C01604 V=800.0 PL=0
MOVL C01605 V=800.0 PL=0
MOVL C01606 V=800.0 PL=0
MOVL C01607 V=800.0 PL=0
MOVL C01608 V=800.0 PL=0
MOVL C01609 V=800.0 PL=0
MOVL C01610 V=800.0 PL=0
MOVL C01611 V=800.0 PL=0
MOVL C01612 V=800.0 PL=0
MOVL C01613 V=800.0 PL=0
MOVL C01614 V=800.0 PL=0
MOVL C01615 V=800.0 PL=0
MOVL C01616 V=800.0 PL=0
MOVL C01617 V=800.0 PL=0
MOVL C01618 V=800.0 PL=0
MOVL C01619 V=800.0 PL=0
MOVL C01620 V=800.0 PL=0
MOVL C01621 V=800.0 PL=0
MOVL C01622 V=800.0 PL=0
MOVL C01623 V=800.0 PL=0
MOVL C01624 V=800.0 PL=0
MOVL C01625 V=800.0 PL=0
MOVL C01626 V=800.0 PL=0
MOVL C01627 V=800.0 PL=0
MOVL C01628 V=800.0 PL=0
MOVL C01629 V=800.0 PL=0
MOVL C01630 V=800.0 PL=0
MOVL C01631 V=800.0 PL=0
MOVL C01632 V=800.0 PL=0
MOVL C01633 V=800.0 PL=0
MOVL C01634 V=800.0 PL=0
MOVL C01635 V=800.0 PL=0
MOVL C01636 V=800.0 PL=0
MOVL C01637 V=800.0 PL=0
MOVL C01638 V=800.0 PL=0
MOVL C01639 V=800.0 PL=0
MOVL C01640 V=800.0 PL=0
MOVL C01641 V=800.0 PL=0
MOVL C01642 V=800.0 PL=0
MOVL C01643 V=800.0 PL=0
MOVL C01644 V=800.0 PL=0
MOVL C01645 V=800.0 PL=0
MOVL C01646 V=800.0 PL=0
MOVL C01647 V=800.0 PL=0
MOVL C01648 V=800.0 PL=0
MOVL C01649 V=800.0 PL=0
MOVL C01650 V=800.0 PL=0
MOVL C01651 V=800.0 PL=0
MOVL C01652 V=800.0 PL=0
MOVL C01653 V=800.0 PL=0
MOVL C01654 V=800.0 PL=0
MOVL C01655 V=800.0 PL=0
MOVL C01656 V=800.0 PL=0
MOVL C01657 V=800.0 PL=0
MOVL C01658 V=800.0 PL=0
MOVL C01659 V=800.0 PL=0
MOVL C01660 V=800.0 PL=0
MOVL C01661 V=800.0 PL=0
MOVL C01662 V=800.0 PL=0
MOVL C01663 V=800.0 PL=0
MOVL C01664 V=800.0 PL=0
MOVL C01665 V=800.0 PL=0
MOVL C01666 V=800.0 PL=0
MOVL C01667 V=800.0 PL=0
MOVL C01668 V=800.0 PL=0
MOVL C01669 V=800.0 PL=0
MOVL C01670 V=800.0 PL=0
MOVL C01671 V=800.0 PL=0
MOVL C01672 V=800.0 PL=0
MOVL C01673 V=800.0 PL=0
MOVL C01674 V=800.0 PL=0
MOVL C01675 V=800.0 PL=0
MOVL C01676 V=800.0 PL=0
MOVL C01677 V=800.0 PL=0
MOVL C01678 V=800.0 PL=0
MOVL C01679 V=800.0 PL=0
MOVL C01680 V=800.0 PL=0
MOVL C01681 V=800.0 PL=0
MOVL C01682 V=800.0 PL=0
MOVL C01683 V=800.0 PL=0
MOVL C01684 V=800.0 PL=0
MOVL C01685 V=800.0 PL=0
MOVL C01686 V=800.0 PL=0
MOVL C01687 V=800.0 PL=0
MOVL C01688 V=800.0 PL=0
MOVL C01689 V=800.0 PL=0
MOVL C01690 V=800.0 PL=0
MOVL C01691 V=800.0 PL=0
MOVL C01692 V=800.0 PL=0
MOVL C01693 V=800.0 PL=0
MOVL C01694 V=800.0 PL=0
MOVL C01695 V=800.0 PL=0
MOVL C01696 V=800.0 PL=0
MOVL C01697 V=800.0 PL=0
MOVL C01698 V=800.0 PL=0
MOVL C01699 V=800.0 PL=0
MOVL C01700 V=800.0 PL=0
MOVL C01701 V=800.0 PL=0
MOVL C01702 V=800.0 PL=0
MOVL C01703 V=800.0 PL=0
MOVL C01704 V=800.0 PL=0
MOVL C01705 V=800.0 PL=0
MOVL C01706 V=800.0 PL=0
MOVL C01707 V=800.0 PL=0
MOVL C01708 V=800.0 PL=0
MOVL C01709 V=800.0 PL=0
MOVL C01710 V=800.0 PL=0
MOVL C01711 V=800.0 PL=0
MOVL C01712 V=800.0 PL=0
MOVL C01713 V=800.0 PL=0
MOVL C01714 V=800.0 PL=0
MOVL C01715 V=800.0 PL=0
MOVL C01716 V=800.0 PL=0
MOVL C01717 V=800.0 PL=0
MOVL C01718 V=800.0 PL=0
MOVL C01719 V=800.0 PL=0
MOVL C01720 V=800.0 PL=0
MOVL C01721 V=800.0 PL=0
MOVL C01722 V=800.0 PL=0
MOVL C01723 V=800.0 PL=0
MOVL C01724 V=800.0 PL=0
MOVL C01725 V=800.0 PL=0
MOVL C01726 V=800.0 PL=0
MOVL C01727 V=800.0 PL=0
MOVL C01728 V=800.0 PL=0
MOVL C01729 V=800.0 PL=0
MOVL C01730 V=800.0 PL=0
MOVL C01731 V=800.0 PL=0
MOVL C01732 V=800.0 PL=0
MOVL C01733 V=800.0 PL=0
MOVL C01734 V=800.0 PL=0
MOVL C01735 V=800.0 PL=0
MOVL C01736 V=800.0 PL=0
MOVL C01737 V=800.0 PL=0
MOVL C01738 V=800.0 PL=0
MOVL C01739 V=800.0 PL=0
MOVL C01740 V=800.0 PL=0
MOVL C01741 V=800.0 PL=0
MOVL C01742 V=800.0 PL=0
MOVL C01743 V=800.0 PL=0
MOVL C01744 V=800.0 PL=0
MOVL C01745 V=800.0 PL=0
MOVL C01746 V=800.0 PL=0
MOVL C01747 V=800.0 PL=0
MOVL C01748 V=800.0 PL=0
MOVL C01749 V=800.0 PL=0
MOVL C01750 V=800.0 PL=0
MOVL C01751 V=800.0 PL=0
MOVL C01752 V=800.0 PL=0
MOVL C01753 V=800.0 PL=0
MOVL C01754 V=800.0 PL=0
MOVL C01755 V=800.0 PL=0
MOVL C01756 V=800.0 PL=0
MOVL C01757 V=800.0 PL=0
MOVL C01758 V=800.0 PL=0
MOVL C01759 V=800.0 PL=0
MOVL C01760 V=800.0 PL=0
MOVL C01761 V=800.0 PL=0
MOVL C01762 V=800.0 PL=0
MOVL C01763 V=800.0 PL=0
MOVL C01764 V=800.0 PL=0
MOVL C01765 V=800.0 PL=0
MOVL C01766 V=800.0 PL=0
MOVL C01767 V=800.0 PL=0
MOVL C01768 V=800.0 PL=0
MOVL C01769 V=800.0 PL=0
MOVL C01770 V=800.0 PL=0
MOVL C01771 V=800.0 PL=0
MOVL C01772 V=800.0 PL=0
MOVL C01773 V=800.0 PL=0
MOVL C01774 V=800.0 PL=0
MOVL C01775 V=800.0 PL=0
MOVL C01776 V=800.0 PL=0
MOVL C01777 V=800.0 PL=0
MOVL C01778 V=800.0 PL=0
MOVL C01779 V=800.0 PL=0
MOVL C01780 V=800.0 PL=0
MOVL C01781 V=800.0 PL=0
MOVL C01782 V=800.0 PL=0
MOVL C01783 V=800.0 PL=0
MOVL C01784 V=800.0 PL=0
MOVL C01785 V=800.0 PL=0
MOVL C01786 V=800.0 PL=0
MOVL C01787 V=800.0 PL=0
MOVL C01788 V=800.0 PL=0
MOVL C01789 V=800.0 PL=0
MOVL C01790 V=800.0 PL=0
MOVL C01791 V=800.0 PL=0
MOVL C01792 V=800.0 PL=0
MOVL C01793 V=800.0 PL=0
MOVL C01794 V=800.0 PL=0
MOVL C01795 V=800.0 PL=0
MOVL C01796 V=800.0 PL=0
MOVL C01797 V=800.0 PL=0
MOVL C01798 V=800.0 PL=0
MOVL C01799 V=800.0 PL=0
MOVL C01800 V=800.0 PL=0
MOVL C01801 V=800.0 PL=0
MOVL C01802 V=800.0 PL=0
MOVL C01803 V=800.0 PL=0
MOVL C01804 V=800.0 PL=0
MOVL C01805 V=800.0 PL=0
MOVL C01806 V=800.0 PL=0
MOVL C01807 V=800.0 PL=0
MOVL C01808 V=800.0 PL=0
MOVL C01809 V=800.0 PL=0
MOVL C01810 V=800.0 PL=0
MOVL C01811 V=800.0 PL=0
MOVL C01812 V=800.0 PL=0
MOVL C01813 V=800.0 PL=0
MOVL C01814 V=800.0 PL=0
MOVL C01815 V=800.0 PL=0
MOVL C01816 V=800.0 PL=0
MOVL C01817 V=800.0 PL=0
MOVL C01818 V=800.0 PL=0
MOVL C01819 V=800.0 PL=0
MOVL C01820 V=800.0 PL=0
MOVL C01821 V=800.0 PL=0
MOVL C01822 V=800.0 PL=0
MOVL C01823 V=800.0 PL=0
MOVL C01824 V=800.0 PL=0
MOVL C01825 V=800.0 PL=0
MOVL C01826 V=800.0 PL=0
MOVL C01827 V=800.0 PL=0
MOVL C01828 V=800.0 PL=0
MOVL C01829 V=800.0 PL=0
MOVL C01830 V=800.0 PL=0
MOVL C01831 V=800.0 PL=0
MOVL C01832 V=800.0 PL=0
MOVL C01833 V=800.0 PL=0
MOVL C01834 V=800.0 PL=0
MOVL C01835 V=800.0 PL=0
MOVL C01836 V=800.0 PL=0
MOVL C01837 V=800.0 PL=0
MOVL C01838 V=800.0 PL=0
MOVL C01839 V=800.0 PL=0
MOVL C01840 V=800.0 PL=0
MOVL C01841 V=800.0 PL=0
MOVL C01842 V=800.0 PL=0
MOVL C01843 V=800.0 PL=0
MOVL C01844 V=800.0 PL=0
MOVL C01845 V=800.0 PL=0
MOVL C01846 V=800.0 PL=0
MOVL C01847 V=800.0 PL=0
MOVL C01848 V=800.0 PL=0
MOVL C01849 V=800.0 PL=0
MOVL C01850 V=800.0 PL=0
MOVL C01851 V=800.0 PL=0
MOVL C01852 V=800.0 PL=0
MOVL C01853 V=800.0 PL=0
MOVL C01854 V=800.0 PL=0
MOVL C01855 V=800.0 PL=0
MOVL C01856 V=800.0 PL=0
MOVL C01857 V=800.0 PL=0
MOVL C01858 V=800.0 PL=0
MOVL C01859 V=800.0 PL=0
MOVL C01860 V=800.0 PL=0
MOVL C01861 V=800.0 PL=0
MOVL C01862 V=800.0 PL=0
MOVL C01863 V=800.0 PL=0
MOVL C01864 V=800.0 PL=0
MOVL C01865 V=800.0 PL=0
MOVL C01866 V=800.0 PL=0
MOVL C01867 V=800.0 PL=0
MOVL C01868 V=800.0 PL=0
MOVL C01869 V=800.0 PL=0
MOVL C01870 V=800.0 PL=0
MOVL C01871 V=800.0 PL=0
MOVL C01872 V=800.0 PL=0
MOVL C01873 V=800.0 PL=0
MOVL C01874 V=800.0 PL=0
MOVL C01875 V=800.0 PL=0
MOVL C01876 V=800.0 PL=0
MOVL C01877 V=800.0 PL=0
MOVL C01878 V=800.0 PL=0
MOVL C01879 V=800.0 PL=0
MOVL C01880 V=800.0 PL=0
MOVL C01881 V=800.0 PL=0
MOVL C01882 V=800.0 PL=0
MOVL C01883 V=800.0 PL=0
MOVL C01884 V=800.0 PL=0
MOVL C01885 V=800.0 PL=0
MOVL C01886 V=800.0 PL=0
MOVL C01887 V=800.0 PL=0
MOVL C01888 V=800.0 PL=0
MOVL C01889 V=800.0 PL=0
MOVL C01890 V=800.0 PL=0
MOVL C01891 V=800.0 PL=0
MOVL C01892 V=800.0 PL=0
MOVL C01893 V=800.0 PL=0
MOVL C01894 V=800.0 PL=0
MOVL C01895 V=800.0 PL=0
MOVL C01896 V=800.0 PL=0
MOVL C01897 V=800.0 PL=0
MOVL C01898 V=800.0 PL=0
MOVL C01899 V=800.0 PL=0
MOVL C01900 V=800.0 PL=0
MOVL C01901 V=800.0 PL=0
MOVL C01902 V=800.0 PL=0
MOVL C01903 V=800.0 PL=0
MOVL C01904 V=800.0 PL=0
MOVL C01905 V=800.0 PL=0
MOVL C01906 V=800.0 PL=0
MOVL C01907 V=800.0 PL=0
MOVL C01908 V=800.0 PL=0
MOVL C01909 V=800.0 PL=0
MOVL C01910 V=800.0 PL=0
MOVL C01911 V=800.0 PL=0
MOVL C01912 V=800.0 PL=0
MOVL C01913 V=800.0 PL=0
MOVL C01914 V=800.0 PL=0
MOVL C01915 V=800.0 PL=0
MOVL C01916 V=800.0 PL=0
MOVL C01917 V=800.0 PL=0
MOVL C01918 V=800.0 PL=0
MOVL C01919 V=800.0 PL=0
MOVL C01920 V=800.0 PL=0
MOVL C01921 V=800.0 PL=0
MOVL C01922 V=800.0 PL=0
MOVL C01923 V=800.0 PL=0
MOVL C01924 V=800.0 PL=0
MOVL C01925 V=800.0 PL=0
MOVL C01926 V=800.0 PL=0
MOVL C01927 V=800.0 PL=0
MOVL C01928 V=800.0 PL=0
MOVL C01929 V=800.0 PL=0
MOVL C01930 V=800.0 PL=0
MOVL C01931 V=800.0 PL=0
MOVL C01932 V=800.0 PL=0
MOVL C01933 V=800.0 PL=0
MOVL C01934 V=800.0 PL=0
MOVL C01935 V=800.0 PL=0
MOVL C01936 V=800.0 PL=0
MOVL C01937 V=800.0 PL=0
MOVL C01938 V=800.0 PL=0
MOVL C01939 V=800.0 PL=0
MOVL C01940 V=800.0 PL=0
MOVL C01941 V=800.0 PL=0
MOVL C01942 V=800.0 PL=0
MOVL C01943 V=800.0 PL=0
MOVL C01944 V=800.0 PL=0
MOVL C01945 V=800.0 PL=0
MOVL C01946 V=800.0 PL=0
MOVL C01947 V=800.0 PL=0
MOVL C01948 V=800.0 PL=0
MOVL C01949 V=800.0 PL=0
MOVL C01950 V=800.0 PL=0
MOVL C01951 V=800.0 PL=0
MOVL C01952 V=800.0 PL=0
MOVL C01953 V=800.0 PL=0
MOVL C01954 V=800.0 PL=0
MOVL C01955 V=800.0 PL=0
MOVL C01956 V=800.0 PL=0
MOVL C01957 V=800.0 PL=0
MOVL C01958 V=800.0 PL=0
MOVL C01959 V=800.0 PL=0
MOVL C01960 V=800.0 PL=0
MOVL C01961 V=800.0 PL=0
MOVL C01962 V=800.0 PL=0
MOVL C01963 V=800.0 PL=0
MOVL C01964 V=800.0 PL=0
MOVL C01965 V=800.0 PL=0
MOVL C01966 V=800.0 PL=0
MOVL C01967 V=800.0 PL=0
MOVL C01968 V=800.0 PL=0
MOVL C01969 V=800.0 PL=0
MOVL C01970 V=800.0 PL=0
MOVL C01971 V=800.0 PL=0
MOVL C01972 V=800.0 PL=0
MOVL C01973 V=800.0 PL=0
MOVL C01974 V=800.0 PL=0
MOVL C01975 V=800.0 PL=0
MOVL C01976 V=800.0 PL=0
MOVL C01977 V=800.0 PL=0
MOVL C01978 V=800.0 PL=0
MOVL C01979 V=800.0 PL=0
MOVL C01980 V=800.0 PL=0
MOVL C01981 V=800.0 PL=0
MOVL C01982 V=800.0 PL=0
MOVL C01983 V=800.0 PL=0
MOVL C01984 V=800.0 PL=0
MOVL C01985 V=800.0 PL=0
MOVL C01986 V=800.0 PL=0
MOVL C01987 V=800.0 PL=0
MOVL C01988 V=800.0 PL=0
MOVL C01989 V=800.0 PL=0
MOVL C01990 V=800.0 PL=0
MOVL C01991 V=800.0 PL=0
MOVL C01992 V=800.0 PL=0
MOVL C01993 V=800.0 PL=0
MOVL C01994 V=800.0 PL=0
MOVL C01995 V=800.0 PL=0
MOVL C01996 V=800.0 PL=0
MOVL C01997 V=800.0 PL=0
MOVL C01998 V=800.0 PL=0
MOVL C01999 V=800.0 PL=0
MOVL C02000 V=800.0 PL=0
MOVL C02001 V=800.0 PL=0
MOVL C02002 V=800.0 PL=0
MOVL C02003 V=800.0 PL=0
MOVL C02004 V=800.0 PL=0
MOVL C02005 V=800.0 PL=0
MOVL C02006 V=800.0 PL=0
MOVL C02007 V=800.0 PL=0
MOVL C02008 V=800.0 PL=0
MOVL C02009 V=800.0 PL=0
MOVL C02010 V=800.0 PL=0
MOVL C02011 V=800.0 PL=0
MOVL C02012 V=800.0 PL=0
MOVL C02013 V=800.0 PL=0
MOVL C02014 V=800.0 PL=0
MOVL C02015 V=800.0 PL=0
MOVL C02016 V=800.0 PL=0
MOVL C02017 V=800.0 PL=0
MOVL C02018 V=800.0 PL=0
MOVL C02019 V=800.0 PL=0
MOVL C02020 V=800.0 PL=0
MOVL C02021 V=800.0 PL=0
MOVL C02022 V=800.0 PL=0
MOVL C02023 V=800.0 PL=0
MOVL C02024 V=800.0 PL=0
MOVL C02025 V=800.0 PL=0
MOVL C02026 V=800.0 PL=0
MOVL C02027 V=800.0 PL=0
MOVL C02028 V=800.0 PL=0
MOVL C02029 V=800.0 PL=0
MOVL C02030 V=800.0 PL=0
MOVL C02031 V=800.0 PL=0
MOVL C02032 V=800.0 PL=0
MOVL C02033 V=800.0 PL=0
MOVL C02034 V=800.0 PL=0
MOVL C02035 V=800.0 PL=0
MOVL C02036 V=800.0 PL=0
MOVL C02037 V=800.0 PL=0
MOVL C02038 V=800.0 PL=0
MOVL C02039 V=800.0 PL=0
MOVL C02040 V=800.0 PL=0
MOVL C02041 V=800.0 PL=0
MOVL C02042 V=800.0 PL=0
MOVL C02043 V=800.0 PL=0
MOVL C02044 V=800.0 PL=0
MOVL C02045 V=800.0 PL=0
MOVL C02046 V=800.0 PL=0
MOVL C02047 V=800.0 PL=0
MOVL C02048 V=800.0 PL=0
MOVL C02049 V=800.0 PL=0
MOVL C02050 V=800.0 PL=0
MOVL C02051 V=800.0 PL=0
MOVL C02052 V=800.0 PL=0
MOVL C02053 V=800.0 PL=0
MOVL C02054 V=800.0 PL=0
MOVL C02055 V=800.0 PL=0
MOVL C02056 V=800.0 PL=0
MOVL C02057 V=800.0 PL=0
MOVL C02058 V=800.0 PL=0
MOVL C02059 V=800.0 PL=0
MOVL C02060 V=800.0 PL=0
MOVL C02061 V=800.0 PL=0
MOVL C02062 V=800.0 PL=0
MOVL C02063 V=800.0 PL=0
MOVL C02064 V=800.0 PL=0
MOVL C02065 V=800.0 PL=0
MOVL C02066 V=800.0 PL=0
MOVL C02067 V=800.0 PL=0
MOVL C02068 V=800.0 PL=0
MOVL C02069 V=800.0 PL=0
MOVL C02070 V=800.0 PL=0
MOVL C02071 V=800.0 PL=0
MOVL C02072 V=800.0 PL=0
MOVL C02073 V=800.0 PL=0
MOVL C02074 V=800.0 PL=0
MOVL C02075 V=800.0 PL=0
MOVL C02076 V=800.0 PL=0
MOVL C02077 V=800.0 PL=0
MOVL C02078 V=800.0 PL=0
MOVL C02079 V=800.0 PL=0
MOVL C02080 V=800.0 PL=0
MOVL C02081 V=800.0 PL=0
MOVL C02082 V=800.0 PL=0
MOVL C02083 V=800.0 PL=0
MOVL C02084 V=800.0 PL=0
MOVL C02085 V=800.0 PL=0
MOVL C02086 V=800.0 PL=0
MOVL C02087 V=800.0 PL=0
MOVL C02088 V=800.0 PL=0
MOVL C02089 V=800.0 PL=0
MOVL C02090 V=800.0 PL=0
MOVL C02091 V=800.0 PL=0
MOVL C02092 V=800.0 PL=0
MOVL C02093 V=800.0 PL=0
MOVL C02094 V=800.0 PL=0
MOVL C02095 V=800.0 PL=0
MOVL C02096 V=800.0 PL=0
MOVL C02097 V=800.0 PL=0
MOVL C02098 V=800.0 PL=0
MOVL C02099 V=800.0 PL=0
MOVL C02100 V=800.0 PL=0
MOVL C02101 V=800.0 PL=0
MOVL C02102 V=800.0 PL=0
MOVL C02103 V=800.0 PL=0
MOVL C02104 V=800.0 PL=0
MOVL C02105 V=800.0 PL=0
MOVL C02106 V=800.0 PL=0
MOVL C02107 V=800.0 PL=0
MOVL C02108 V=800.0 PL=0
MOVL C02109 V=800.0 PL=0
MOVL C02110 V=800.0 PL=0
MOVL C02111 V=800.0 PL=0
MOVL C02112 V=800.0 PL=0
MOVL C02113 V=800.0 PL=0
MOVL C02114 V=800.0 PL=0
MOVL C02115 V=800.0 PL=0
MOVL C02116 V=800.0 PL=0
MOVL C02117 V=800.0 PL=0
MOVL C02118 V=800.0 PL=0
MOVL C02119 V=800.0 PL=0
MOVL C02120 V=800.0 PL=0
MOVL C02121 V=800.0 PL=0
MOVL C02122 V=800.0 PL=0
MOVL C02123 V=800.0 PL=0
MOVL C02124 V=800.0 PL=0
MOVL C02125 V=800.0 PL=0
MOVL C02126 V=800.0 PL=0
MOVL C02127 V=800.0 PL=0
MOVL C02128 V=800.0 PL=0
MOVL C02129 V=800.0 PL=0
MOVL C02130 V=800.0 PL=0
MOVL C02131 V=800.0 PL=0
MOVL C02132 V=800.0 PL=0
